	(* PINZA: ASPIRAZIONE/APERTURA CHIUSURA *)
	IF ManCmdJHomeTRIG AND MachinePalletizer_TF.Modules^.AX_J.CmdExe.Code = CmdNOP THEN
		ManCmdJHomeTRIG := FALSE;
	END_IF
	IF MachinePalletizer_TF.ManCmd^.Pinza.ApriPinza THEN
		TFParametersArrayClear(ADR(ParametersArray));
		ParametersArray.Parameters[0] := '1';
		ParametersArray.Parameters[1] := '10';
		TFCommandSend(CmdMAN,ParametersArray,MachinePalletizer_TF.Modules^.Pinza.Cmd);
		MachinePalletizer_TF.ManCmd^.Pinza.ApriPinza := FALSE;
	END_IF
	IF MachinePalletizer_TF.ManCmd^.Pinza.ChiudiPinza THEN
		TFParametersArrayClear(ADR(ParametersArray));
		ParametersArray.Parameters[0] := '1';
		ParametersArray.Parameters[1] := '11';
		MachinePalletizer_TF.ManCmd^.Pinza.ChiudiPinza := FALSE;
		TFCommandSend(CmdMAN,ParametersArray,MachinePalletizer_TF.Modules^.Pinza.Cmd);
	END_IF
	IF MachinePalletizer_TF.ManCmd^.Pinza.SbloccoPinza THEN
		TFParametersArrayClear(ADR(ParametersArray));
		ParametersArray.Parameters[0] := '1';
		ParametersArray.Parameters[1] := '20';
		MachinePalletizer_TF.ManCmd^.Pinza.SbloccoPinza:= FALSE;
		TFCommandSend(CmdMAN,ParametersArray,MachinePalletizer_TF.Modules^.Pinza.Cmd);
	END_IF
	IF MachinePalletizer_TF.ManCmd^.Pinza.BloccoPinza THEN
		TFParametersArrayClear(ADR(ParametersArray));
		ParametersArray.Parameters[0] := '1';
		ParametersArray.Parameters[1] := '21';
		MachinePalletizer_TF.ManCmd^.Pinza.BloccoPinza:= FALSE;
		TFCommandSend(CmdMAN,ParametersArray,MachinePalletizer_TF.Modules^.Pinza.Cmd);
	END_IF
	IF MachinePalletizer_TF.ManCmd^.Pinza.AttivazioneVuotoFaldeDX THEN
		TFParametersArrayClear(ADR(ParametersArray));
		ParametersArray.Parameters[0] := '1';
		ParametersArray.Parameters[1] := '30';
		MachinePalletizer_TF.ManCmd^.Pinza.AttivazioneVuotoFaldeDX := FALSE;
		TFCommandSend(CmdMAN,ParametersArray,MachinePalletizer_TF.Modules^.Pinza.Cmd);
	END_IF
	IF MachinePalletizer_TF.ManCmd^.Pinza.DisattivazioneVuotoFaldeDX THEN
		TFParametersArrayClear(ADR(ParametersArray));
		ParametersArray.Parameters[0] := '1';
		ParametersArray.Parameters[1] := '31';
		MachinePalletizer_TF.ManCmd^.Pinza.DisattivazioneVuotoFaldeDX := FALSE;
		TFCommandSend(CmdMAN,ParametersArray,MachinePalletizer_TF.Modules^.Pinza.Cmd);
	END_IF
	IF MachinePalletizer_TF.ManCmd^.Pinza.AttivazioneVuotoFaldeSX THEN
		TFParametersArrayClear(ADR(ParametersArray));
		ParametersArray.Parameters[0] := '1';
		ParametersArray.Parameters[1] := '40';
		MachinePalletizer_TF.ManCmd^.Pinza.AttivazioneVuotoFaldeSX := FALSE;
		TFCommandSend(CmdMAN,ParametersArray,MachinePalletizer_TF.Modules^.Pinza.Cmd);
	END_IF
	IF MachinePalletizer_TF.ManCmd^.Pinza.DisattivazioneVuotoFaldeSX THEN
		TFParametersArrayClear(ADR(ParametersArray));
		ParametersArray.Parameters[0] := '1';
		ParametersArray.Parameters[1] := '41';
		MachinePalletizer_TF.ManCmd^.Pinza.DisattivazioneVuotoFaldeSX := FALSE;
		TFCommandSend(CmdMAN,ParametersArray,MachinePalletizer_TF.Modules^.Pinza.Cmd);
	END_IF
	IF MachinePalletizer_TF.ManCmd^.Pinza.AttivazioneVuotoDX THEN
		TFParametersArrayClear(ADR(ParametersArray));
		ParametersArray.Parameters[0] := '1';
		ParametersArray.Parameters[1] := '50';
		MachinePalletizer_TF.ManCmd^.Pinza.AttivazioneVuotoDX := FALSE;
		TFCommandSend(CmdMAN,ParametersArray,MachinePalletizer_TF.Modules^.Pinza.Cmd);
	END_IF
//	IF MachinePalletizer_TF.ManCmd^.Pinza.DisattivazioneVuotoDX THEN
//		TFParametersArrayClear(ADR(ParametersArray));
//		ParametersArray.Parameters[0] := '1';
//		ParametersArray.Parameters[1] := '51';
//		MachinePalletizer_TF.ManCmd^.Pinza.DisattivazioneVuotoDX := FALSE;
//		TFCommandSend(CmdMAN,ParametersArray,MachinePalletizer_TF.Modules^.Pinza.Cmd);
//	END_IF
	IF MachinePalletizer_TF.ManCmd^.Pinza.AttivazioneVuotoSX THEN
		TFParametersArrayClear(ADR(ParametersArray));
		ParametersArray.Parameters[0] := '1';
		ParametersArray.Parameters[1] := '60';
		MachinePalletizer_TF.ManCmd^.Pinza.AttivazioneVuotoSX := FALSE;
		TFCommandSend(CmdMAN,ParametersArray,MachinePalletizer_TF.Modules^.Pinza.Cmd);
	END_IF
	IF MachinePalletizer_TF.ManCmd^.Pinza.DisattivazioneVuotoSX THEN
		
		IF Ciclo_Deposito_Lastra.Stato <> ANNULLATO AND NOT EseguitoAllinementoPezziDeposito(*AND MachinePalletizer_TF.Modules^.Pinza.AspirazioneSX^.Out.Attiva_Vuoto AND MachinePalletizer_TF.Modules^.Pinza.StatoPinza.LatoSxPiastrellaInPresa*) THEN
			IF Mission.PPlace > 0 THEN
				//Aggiungo la lastra in deposito e aggiorno lo stato della lastra della lista in modo da contrasegnarla elaborata 
				IF (MachinePalletizerModules.AX_X.Ax^.AxRef^.NcToPlc.ActPos >= WorkArea[Mission.PPlace].X - 300) AND 
					(MachinePalletizerModules.AX_X.Ax^.AxRef^.NcToPlc.ActPos <= WorkArea[Mission.PPlace].X + 300) THEN
					//WorkAreaState[Mission.PPlace].Slab[WorkAreaState[Mission.PPlace].P] 	:= MachinePalletizerModules.Pinza.ElementoInPrelievo^;
					//WorkAreaState[Mission.PPlace].SlabData[WorkAreaState[Mission.PPlace].P] := MachinePalletizerModules.Pinza.DataElement^;
					WorkAreaState[Mission.PPlace].P := WorkAreaState[Mission.PPlace].P +1;
					HMI_NumeroPezziPresentiPostazione[Mission.PPlace] := HMI_NumeroPezziPresentiPostazione[Mission.PPlace] + 1;
					FOR i := 1 TO MAXELEMENTLIST DO
						IF WorkAreaProductionList[Mission.PPlace].PElementList[i].Stato = ELEMENTO_DA_ELABORARE THEN
							WorkAreaProductionList[Mission.PPlace].PElementList[i].Stato := ELEMENTO_ELABORATO; //Dichiaro che l'elemento della lista è stato elaborato
							EXIT;
						END_IF
					END_FOR	
					EseguitoAllinementoPezziDeposito := TRUE;				
				ELSE
					;
				END_IF
				//aggiungo nel prelievo la lastra se è stata rimessa al suo posto
				IF (MachinePalletizerModules.AX_X.Ax^.AxRef^.NcToPlc.ActPos >= WorkArea[Mission.PPick].X - 300) AND 
					(MachinePalletizerModules.AX_X.Ax^.AxRef^.NcToPlc.ActPos <= WorkArea[Mission.PPick].X + 300) THEN
					//WorkAreaState[Mission.PPlace].Slab[WorkAreaState[Mission.PPlace].P] 	:= MachinePalletizerModules.Pinza.ElementoInPrelievo^;
					//WorkAreaState[Mission.PPlace].SlabData[WorkAreaState[Mission.PPlace].P] := MachinePalletizerModules.Pinza.DataElement^;
					WorkAreaState[Mission.PPick].P := WorkAreaState[Mission.PPick].P +1;
					HMI_NumeroPezziPresentiPostazione[Mission.PPick] := HMI_NumeroPezziPresentiPostazione[Mission.PPick] + 1;
					EseguitoAllinementoPezziDeposito := TRUE;	
				ELSE
					;
				END_IF
			END_IF
			
		END_IF
	
		TFParametersArrayClear(ADR(ParametersArray));
		ParametersArray.Parameters[0] := '1';
		ParametersArray.Parameters[1] := '61';
		MachinePalletizer_TF.ManCmd^.Pinza.DisattivazioneVuotoSX := FALSE;
		TFCommandSend(CmdMAN,ParametersArray,MachinePalletizer_TF.Modules^.Pinza.Cmd);
		Ciclo_Prelievo_Lastra.Stato 		:= ANNULLATO;
		Ciclo_Pelievo_Falda.Stato 			:= ANNULLATO;
		Ciclo_Deposito_Lastra.Stato			:= ANNULLATO;
		Ciclo_Deposito_Falda.Stato			:= ANNULLATO;
		Ciclo_Di_Riposo.Stato				:= ANNULLATO;
		Ciclo_Prelievo_Lastra_Depal.Stato 	:= ANNULLATO;
		Ciclo_Deposito_Lastra_Depal.Stato 	:= ANNULLATO;
		Ciclo_Deposito_Falda_Depal.Stato 	:= ANNULLATO;
		ProductOnGripper 					:= KNOPRODUCT;
		Ciclo_Deposito_Falda_Depal.Stato 	:= ANNULLATO;
		
		//Azzero hli apprendimenti e riporto le quote allo stato iniziale
		FOR i:=1 TO MAXAREAPRESENT DO
			WorkAreaState[i].Apprendimento.Z.Lato0.Stato 	:= APPRENDIMENTO_DA_ESEGUIRE;
			WorkAreaState[i].Apprendimento.Z.Lato90.Stato 	:= APPRENDIMENTO_DA_ESEGUIRE;
			WorkAreaState[i].Apprendimento.Z.Lato180.Stato 	:= APPRENDIMENTO_DA_ESEGUIRE;
		END_FOR
		
		StatoMissione 				:= MISSION_STATE_NOP;//Azzero segnalazione a HMI
		WorkAreaManager.State 		:= WAMANAGER_NOP;
		Mission.State 				:= MISSION_STATE_NOP;
		MaterialeDepositatoSuLinea 	:= TRUE;//In questo modo se scarico la mattonella sulla rulliera, lei parte
	END_IF
	IF MachinePalletizer_TF.ManCmd^.Pinza.AttivaTastatori THEN
		TFParametersArrayClear(ADR(ParametersArray));
		ParametersArray.Parameters[0] := '1';
		ParametersArray.Parameters[1] := '70';
		MachinePalletizer_TF.ManCmd^.Pinza.AttivaTastatori := FALSE;
		TFCommandSend(CmdMAN,ParametersArray,MachinePalletizer_TF.Modules^.Pinza.Cmd);
	END_IF
	IF MachinePalletizer_TF.ManCmd^.Pinza.DisattivaTastatori THEN
		TFParametersArrayClear(ADR(ParametersArray));
		ParametersArray.Parameters[0] := '1';
		ParametersArray.Parameters[1] := '71';
		MachinePalletizer_TF.ManCmd^.Pinza.DisattivaTastatori := FALSE;
		TFCommandSend(CmdMAN,ParametersArray,MachinePalletizer_TF.Modules^.Pinza.Cmd);
	END_IF
	IF MachinePalletizer_TF.ManCmd^.Pinza.CalibrazioneOVEM THEN
		TFParametersArrayClear(ADR(ParametersArray));
		MachinePalletizer_TF.ManCmd^.Pinza.CalibrazioneOVEM := FALSE;
		TFCommandSend(CmdHOME,ParametersArray,MachinePalletizer_TF.Modules^.Pinza.Cmd);
	END_IF

	//Posizionamento diretto pinza
	IF MachinePalletizer_TF.ManCmd^.PosizionamentoPinza0 THEN
		TFParametersArrayClear(ADR(ParametersArray));
		ParametersArray.Parameters[0] := '100';
		ParametersArray.Parameters[1] := '13';
		MachinePalletizer_TF.Modules^.AX_J.AxisPar^.Quota_Destinazione := 0;
		TFCommandSend(CmdMAN,ParametersArray,MachinePalletizer_TF.Modules^.AX_J.Cmd);
		MachinePalletizer_TF.ManCmd^.PosizionamentoPinza0 := FALSE;
	END_IF
	IF MachinePalletizer_TF.ManCmd^.PosizionamentoPinza90 THEN
		TFParametersArrayClear(ADR(ParametersArray));
		ParametersArray.Parameters[0] := '100';
		ParametersArray.Parameters[1] := '13';
		MachinePalletizer_TF.Modules^.AX_J.AxisPar^.Quota_Destinazione := 90;
		TFCommandSend(CmdMAN,ParametersArray,MachinePalletizer_TF.Modules^.AX_J.Cmd);
		 MachinePalletizer_TF.ManCmd^.PosizionamentoPinza90 := FALSE;
	END_IF
	IF MachinePalletizer_TF.ManCmd^.PosizionamentoPinza180 THEN
		TFParametersArrayClear(ADR(ParametersArray));
		ParametersArray.Parameters[0] := '100';
		ParametersArray.Parameters[1] := '13';
		MachinePalletizer_TF.Modules^.AX_J.AxisPar^.Quota_Destinazione := 180;
		TFCommandSend(CmdMAN,ParametersArray,MachinePalletizer_TF.Modules^.AX_J.Cmd);
		MachinePalletizer_TF.ManCmd^.PosizionamentoPinza180 := FALSE;
	END_IF
	
	IF ManCmdXHomeTRIG AND 
		MachinePalletizer_TF.Modules^.AX_X.CmdExe.Code = CmdNOP THEN
		ManCmdXHomeTRIG := FALSE;
		MachinePalletizer_TF.ManCmd^.X.Home:= FALSE;
	END_IF
	IF ManCmdYHomeTRIG AND 
		MachinePalletizer_TF.Modules^.AX_Y.CmdExe.Code = CmdNOP THEN
		ManCmdYHomeTRIG := FALSE;
		MachinePalletizer_TF.ManCmd^.Y.Home:= FALSE;
	END_IF
	IF ManCmdZHomeTRIG AND 
		MachinePalletizer_TF.Modules^.AX_Z.CmdExe.Code = CmdNOP THEN
		ManCmdZHomeTRIG := FALSE;
		MachinePalletizer_TF.ManCmd^.Z.Home:= FALSE;
	END_IF
	IF ManCmdJHomeTRIG AND 
		MachinePalletizer_TF.Modules^.AX_J.CmdExe.Code = CmdNOP THEN
		ManCmdJHomeTRIG := FALSE;
		MachinePalletizer_TF.ManCmd^.J.Home:= FALSE;
	END_IF
	
END_IF
END_ACTION

ACTION _06_ScriviOutput:
(* Control Word OVEM *)
O_ControlWordOVEM_1 := MachinePalletizerModules.Pinza.AspirazioneDX1^.Out.ControlWord;
O_ControlWordOVEM_2 := MachinePalletizerModules.Pinza.AspirazioneSX1^.Out.ControlWord;

O_ControlWordOVEM_12 := MachinePalletizerModules.Pinza.AspirazioneDX2^.Out.ControlWord;
O_ControlWordOVEM_22 := MachinePalletizerModules.Pinza.AspirazioneSX2^.Out.ControlWord;

(* Configurazione Porte Ciabatta Pinza *)

{info 'TODO:SISTEMARE IO PINZA'}	

//Q_K517[22] := 1; //Configurazione pin 2 e pin 4 come uscite porta X1.0
//Q_K517[23] := 1; //Configurazione pin 2 e pin 4 come uscite porta X1.1
//Q_K517[24] := 1; //Configurazione pin 2 e pin 4 come uscite porta X1.2
Q_K517[25] := 1; //Configurazione pin 2 e pin 4 come uscite porta X1.3
//Q_K517[26] := 1; //Configurazione pin 2 e pin 4 come uscite porta X1.4
//Q_K517[27] := 1; //Configurazione pin 2 e pin 4 come uscite porta X1.5
Q_K517[28] := 1; //Configurazione pin 2 e pin 4 come uscite porta X1.6
Q_K517[29] := 1; //Configurazione pin 2 e pin 4 come uscite porta X1.7

//Q_K517[2].0 //Comando X1.0 pin 4
//Q_K517[2].1 //Comando X1.1 pin 4
//Q_K517[2].2 //Comando X1.2 pin 4
//Q_K517[2].3 //Comando X1.3 pin 4
//Q_K517[2].4 //Comando X1.4 pin 4
//Q_K517[2].5 //Comando X1.5 pin 4
//Q_K517[2].6 //Comando X1.6 pin 4
//Q_K517[2].7 //Comando X1.7 pin 4
///------------------------------//
//Q_K517[3].0 //Comando X1.0 pin 2
//Q_K517[3].1 //Comando X1.1 pin 2
//Q_K517[3].2 //Comando X1.2 pin 2
//Q_K517[3].3 //Comando X1.3 pin 2
//Q_K517[3].4 //Comando X1.4 pin 2
//Q_K517[3].5 //Comando X1.5 pin 2
//Q_K517[3].6 //Comando X1.6 pin 2
//Q_K517[3].7 //Comando X1.7 pin 2

Q_K517[2].3 := MachinePalletizerModules.Pinza.AspirazioneFaldaDX^.OUT.ActivationOutput;
Q_K517[2].6 := MachinePalletizerModules.Pinza.CilindroSbloccoBascolante^.OUT.ActivationOutput;
Q_K517[2].7 := MachinePalletizerModules.Pinza.CilindroSbloccoRotazione^.OUT.ActivationOutput;

//Q_J17[3].7 := MachinePalletizerModules.Pinza.CilindroTasteggio^.OUT.ActivationOutput;

LetturaFTCPinza0_1 		:= MachinePalletizerModules.Pinza.StatoPinza.LetturaFTC0;
LetturaFTCPinza180_1 	:= MachinePalletizerModules.Pinza.StatoPinza.LetturaFTC180;
LetturaFTCPinza0_2 		:= MachinePalletizerModules.Pinza.StatoPinza.LetturaFTC0_2;
LetturaFTCPinza180_2 	:= MachinePalletizerModules.Pinza.StatoPinza.LetturaFTC180_2;

(* ******************************************************************************************************** *)
(* OUTPUT Transfer *)
(* ******************************************************************************************************** *)

(* Pallet and Layer stacks state *)
PalletStackEmpty 												:= MachinePalletizer_TF.PalletStackEmpty;
LayerStackEmpty 												:= MachinePalletizer_TF.LayerStackEmpty;
AllWABusy 														:= MachinePalletizer_TF.AllWABusy;

(* Machine Palletizer *)
O_ResetACKAzionamenti 	:= I_StartCicloPal OR MachinePalletizerGatesAccess.GateAccessConsolle.ErrAckDriver;// OR MachinePalletizerGatesAccess.GateAccess2.ErrAckDriver;// OR MachinePalletizerLGV.ErrAckDriver;
O_AbilitazioneMarcia	:= MachinePalletizer_TF.OUT.PowerActive;


O_SirenaAllarmiPal		:= MachinePalletizer_TF.OUT.StartHorn OR MachinePalletizer_TF.OUT.Horn OR (MachinePalletizer_TF.OUT.Warning AND MachinePalletizer_TF.OUT.ClockSegnalazioniAlternato AND NOT MachinePalletizer_TF.OUT.ResetSirenaSegnalazioni);// OR (I_Trasporti_GEN_GLOBAL_ALARM_STOP AND MachinePalletizer_TF.OUT.ClockSegnalazioni);

O_LampadaAutomaticoPal	:= MachinePalletizer_TF.OUT.Run;

O_LampadaAllarmiPal		:= (MachinePalletizer_TF.OUT.Error AND MachinePalletizer_TF.OUT.ClockSegnalazioni) OR
							MachinePalletizer_TF.OUT.Error;
							
																	
O_Reset_Plc_Sicurezza := I_StartCicloPal OR 
						MachinePalletizerGatesAccess.GateAccessConsolle.ErrAck OR
						MachinePalletizerGatesAccess.GateAccessPS306.ErrAck OR
						MachinePalletizerGatesAccess.GateAccessPS307.ErrAck OR
						MachinePalletizerGatesAccess.GateAccessPS308.ErrAck OR
						MachinePalletizerGatesAccess.GateAccessPS309.ErrAck;


O_LampadaPulsanteCicloPalConsolle:= MachinePalletizer_TF.OUT.Run OR 
									(ResetNecessarioCentralinaSafety AND MachinePalletizer_TF.OUT.ClockSegnalazioni) ;
O_LampadaPulsanteMarciaPalConsolle := I_MarciaOK AND (MachinePalletizerModules.AX_X.Ax^.Status.PowerActive AND 
													MachinePalletizerModules.AX_Y.Ax^.Status.PowerActive AND 
													MachinePalletizerModules.AX_Z.Ax^.Status.PowerActive AND 
													MachinePalletizerModules.AX_J.Ax^.Status.PowerActive) OR 
										((I_MarciaOK AND NOT(MachinePalletizerModules.AX_X.Ax^.Status.PowerActive AND 
														MachinePalletizerModules.AX_Y.Ax^.Status.PowerActive AND 
														MachinePalletizerModules.AX_Z.Ax^.Status.PowerActive AND 
														MachinePalletizerModules.AX_J.Ax^.Status.PowerActive) OR
										(I_SafetyStateEmergenze_Generali <> 1 OR 
                                          I_SafetyStateEmergenza_PS306_307 <> 1 OR
                                          I_SafetyStateEmergenza_PS308_309 <> 1)) AND MachinePalletizer_TF.OUT.ClockSegnalazioni)AND NOT ResetNecessarioCentralinaSafety;

(* Gates Access *)
O_LampadaRichiestaIngressoPal	:= (MachinePalletizerGatesAccess.GateAccessConsolle.AccessLamp OR 
									MachinePalletizerGatesAccess.GateAccessPS306.AccessLamp OR
									MachinePalletizerGatesAccess.GateAccessPS307.AccessLamp OR 
									MachinePalletizerGatesAccess.GateAccessPS308.AccessLamp OR 
									MachinePalletizerGatesAccess.GateAccessPS309.AccessLamp OR
									(NOT I_BarrierePallettizzatoreOK AND MachinePalletizer_TF.OUT.ClockSegnalazioni))AND NOT ResetNecessarioCentralinaSafety;

O_LampadaPulsanteRichiestaIngressoConsolle := MachinePalletizerGatesAccess.GateAccessConsolle.AccessLamp OR 
											((I_BarrierePallettizzatoreOK <> 1 AND MachinePalletizer_TF.OUT.ClockSegnalazioni) AND NOT ResetNecessarioCentralinaSafety);
									
O_LampadaPulsanteRichiestaIngressoPS306 := MachinePalletizerGatesAccess.GateAccessPS306.AccessLamp OR 
											((NOT I_BarrierePallettizzatoreOK AND MachinePalletizer_TF.OUT.ClockSegnalazioni) AND NOT ResetNecessarioCentralinaSafety);

O_LampadaPulsanteRichiestaIngressoPS307 := MachinePalletizerGatesAccess.GateAccessPS307.AccessLamp OR 
											((NOT I_BarrierePallettizzatoreOK AND MachinePalletizer_TF.OUT.ClockSegnalazioni) AND NOT ResetNecessarioCentralinaSafety);

O_LampadaPulsanteRichiestaIngressoPS308 := MachinePalletizerGatesAccess.GateAccessPS308.AccessLamp OR 
											((NOT I_BarrierePallettizzatoreOK AND MachinePalletizer_TF.OUT.ClockSegnalazioni) AND NOT ResetNecessarioCentralinaSafety);

O_LampadaPulsanteRichiestaIngressoPS309 := MachinePalletizerGatesAccess.GateAccessPS309.AccessLamp OR 
											((NOT I_BarrierePallettizzatoreOK AND MachinePalletizer_TF.OUT.ClockSegnalazioni) AND NOT ResetNecessarioCentralinaSafety);
									
//******************** SCHEDA OUT AP201.4
O_AP201_4[1]	:= O_SirenaAllarmiPal;				
O_AP201_4[2]	:= O_LampadaAutomaticoPal;			
O_AP201_4[3]	:= O_LampadaAllarmiPal;				
O_AP201_4[4]	:= O_LampadaRichiestaIngressoPal;
O_AP201_4[5]	:= O_ConsensoVeicolo[1];						
O_AP201_4[6]	:= O_ConsensoVeicolo[2];						
O_AP201_4[7]	:= O_ConsensoVeicolo[3];						
O_AP201_4[8]	:= O_ConsensoVeicolo[4];						
O_AP201_4[9]	:= O_LampadaPulsanteCicloPalConsolle; 			
O_AP201_4[10]	:= O_LampadaPulsanteRichiestaIngressoConsolle; 	
O_AP201_4[11]	:= O_LampadaPulsanteMarciaPalConsolle;			
O_AP201_4[12]	:= O_LampadaPulsanteRichiestaIngressoPS306; 	
O_AP201_4[13]	:= O_LampadaPulsanteRichiestaIngressoPS307;		
O_AP201_4[14]	:= O_LampadaPulsanteRichiestaIngressoPS308; 	
O_AP201_4[15]	:= O_LampadaPulsanteRichiestaIngressoPS309;		
O_AP201_4[16]	:= FALSE; 										
											
//******************** SCHEDA OUT SAFETY AP201.5											
O_AP201_5;											
//O_MarciaPal	: BOOL; // CH1=											
//FREE			: BOOL; // CH2=												
//FREE			: BOOL; // CH3=												
//FREE			: BOOL; // CH4=			
									
//******************** SCHEDA OUT AP201.6												
O_AP201_6[1]	:= O_LampadaIngressoVietatoPS306; 												
O_AP201_6[2]	:= O_LampadaIngressoVietatoPS307; 												
O_AP201_6[3]	:= O_LampadaIngressoVietatoPS308; 												
O_AP201_6[4]	:= O_LampadaIngressoVietatoPS309; 												
O_AP201_6[5]	:= O_ConsensoVeicolo[5];		  												
O_AP201_6[6]	:= O_ConsensoVeicolo[6];														
O_AP201_6[7]	:= O_ConsensoVeicolo[7];														
O_AP201_6[8]	:= O_ConsensoVeicolo[8];														
O_AP201_6[9]	:= FALSE; 																		
O_AP201_6[10]	:= FALSE; 																		
O_AP201_6[11]	:= FALSE; 																		
O_AP201_6[12]	:= FALSE; 																		
O_AP201_6[13]	:= FALSE; 																		
O_AP201_6[14]	:= FALSE; 							
O_AP201_6[15]	:= FALSE; 							
O_AP201_6[16]	:= FALSE; 							


O_XDriveDigitalOutput.1 := O_SbloccoFermoSicurezza; //Sblocco del paracadute -> ingresso 1 del drive X
END_ACTION

ACTION _07_ScriviStatus:
(*Valorizzazione della struttura Status_TF*)

(*Stato Macchina*)
Status_TF.Macchina.Auto					:= MachinePalletizer_TF.IN.Mode.Auto AND MachinePalletizer_TF.CmdExe.Code = CmdDO;
Status_TF.Macchina.Run					:= MachinePalletizer_TF.OUT.Run;
Status_TF.Macchina.Error				:= MachinePalletizer_TF.Error.Code;
Status_TF.Macchina.ErrorExtra			:= MachinePalletizer_TF.Error.ExtraCode;
Status_TF.Macchina.PowerOK				:= MachinePalletizer_TF.IN.PowerOk;
Status_TF.Macchina.EmergencyOK			:= MachinePalletizer_TF.IN.Mode.EmergencyRequest;

(*Stato assi*)	
Status_TF.X.Position 					:= MachinePalletizerModules.AX_X.Ax^.Status.ActPosition;
Status_TF.X.Velocity 					:= MachinePalletizerModules.AX_X.Ax^.Status.ActVelocity;
Status_TF.X.Torque 						:= MachinePalletizerModules.AX_X.Ax^.Status.ActTorque;
Status_TF.X.Error 						:= MachinePalletizerModules.AX_X.Ax^.Status.ErrorID;
Status_TF.X.PowerActive					:= MachinePalletizerModules.AX_X.Ax^.Status.PowerActive;

Status_TF.Y.Position 					:= MachinePalletizerModules.AX_Y.Ax^.Status.ActPosition;
Status_TF.Y.Velocity 					:= MachinePalletizerModules.AX_Y.Ax^.Status.ActVelocity;
Status_TF.Y.Torque 						:= MachinePalletizerModules.AX_Y.Ax^.Status.ActTorque;
Status_TF.Y.Error 						:= MachinePalletizerModules.AX_Y.Ax^.Status.ErrorID;
Status_TF.Y.PowerActive					:= MachinePalletizerModules.AX_Y.Ax^.Status.PowerActive;

Status_TF.Z.Position 					:= MachinePalletizerModules.AX_Z.Ax^.Status.ActPosition;
Status_TF.Z.Velocity 					:= MachinePalletizerModules.AX_Z.Ax^.Status.ActVelocity;
Status_TF.Z.Torque 						:= MachinePalletizerModules.AX_Z.Ax^.Status.ActTorque;
Status_TF.Z.Error 						:= MachinePalletizerModules.AX_Z.Ax^.Status.ErrorID;
Status_TF.Z.PowerActive					:= MachinePalletizerModules.AX_Z.Ax^.Status.PowerActive;

Status_TF.J.Position 					:= MachinePalletizerModules.AX_J.Ax^.Status.ActPosition;
Status_TF.J.Velocity 					:= MachinePalletizerModules.AX_J.Ax^.Status.ActVelocity;
Status_TF.J.Torque 						:= MachinePalletizerModules.AX_J.Ax^.Status.ActTorque;
Status_TF.J.Error 						:= MachinePalletizerModules.AX_J.Ax^.Status.ErrorID;
Status_TF.J.PowerActive					:= MachinePalletizerModules.AX_J.Ax^.Status.PowerActive;

Status_TF.K.Position 					:= 0;//ModuloAsse_K.Ax^.Status.ActPosition;
Status_TF.K.Velocity 					:= 0;//ModuloAsse_K.Ax^.Status.ActVelocity;
Status_TF.K.Torque 						:= 0;//ModuloAsse_K.Ax^.Status.ActTorque;
Status_TF.K.Error 						:= 0;//ModuloAsse_K.Ax^.Status.ErrorID;
Status_TF.K.PowerActive					:= 0;//ModuloAsse_K.Ax^.Status.PowerActive;

(*Stato Moduli*)
//Status_TF.ModAsse_X.Cmd					:= ModuloAsse_X.CmdExe.Code;
//Status_TF.ModAsse_X.CmdCase				:= ModuloAsse_X.CmdExe.CmdCase;
Status_TF.ModAsse_X.Error       		:= MachinePalletizerModules.AX_X.Error.Code;
Status_TF.ModAsse_X.ErrorExtra      	:= MachinePalletizerModules.AX_X.Error.ExtraCode;

//Status_TF.ModAsse_Y.Cmd					:= ModuloAsse_Y.CmdExe.Code;
//Status_TF.ModAsse_Y.CmdCase				:= ModuloAsse_Y.CmdExe.CmdCase;
Status_TF.ModAsse_Y.Error       		:= MachinePalletizerModules.AX_Y.Error.Code;
Status_TF.ModAsse_Y.ErrorExtra      	:= MachinePalletizerModules.AX_Y.Error.ExtraCode;

//Status_TF.ModAsse_Z.Cmd					:= ModuloAsse_Z.CmdExe.Code;
//Status_TF.ModAsse_Z.CmdCase				:= ModuloAsse_Z.CmdExe.CmdCase;
Status_TF.ModAsse_Z.Error       		:= MachinePalletizerModules.AX_Z.Error.Code;
Status_TF.ModAsse_Z.ErrorExtra      	:= MachinePalletizerModules.AX_Z.Error.ExtraCode;

//Status_TF.ModAsse_J.Cmd					:= ModuloAsse_J.CmdExe.Code;
//Status_TF.ModAsse_J.CmdCase				:= ModuloAsse_J.CmdExe.CmdCase;
Status_TF.ModAsse_J.Error       		:= MachinePalletizerModules.AX_J.Error.Code;
Status_TF.ModAsse_J.ErrorExtra      	:= MachinePalletizerModules.AX_J.Error.ExtraCode;

//Status_TF.ModAsse_K.Cmd					:= ModuloAsse_K.CmdExe.Code;
//Status_TF.ModAsse_K.CmdCase				:= ModuloAsse_K.CmdExe.CmdCase;
Status_TF.ModAsse_K.Error       		:= 0;//ModuloAsse_K.Error.Code;
Status_TF.ModAsse_K.ErrorExtra      	:= 0;//ModuloAsse_K.Error.ExtraCode;

//Status_TF.ModAspirazione.Cmd			:= ModuloAspirazione.CmdExe.Code;
//Status_TF.ModAspirazione.CmdCase		:= ModuloAspirazione.CmdExe.CmdCase;
Status_TF.ModAspirazione.Error       	:= MachinePalletizerModules.Pinza.Error.Code;
Status_TF.ModAspirazione.ErrorExtra     := MachinePalletizerModules.Pinza.Error.ExtraCode;

Status_TF.Pinza.Module.Error       	:= MachinePalletizerModules.Pinza.Error.Code;
Status_TF.Pinza.Module.ErrorExtra     := MachinePalletizerModules.Pinza.Error.ExtraCode;


(* Trsferimento a Struttura dati Creo *)
Status.MachineAuto := Status_TF.Macchina.Auto;
Status.MachineError := Status_TF.Macchina.Error;
Status.MachineErrorExtra := Status_TF.Macchina.ErrorExtra;

//Pinza Cilindro Cilindro Aspirazione DX
Status_TF.Pinza.AspirazioneDX.Active 			:= MachinePalletizerModules.Pinza.AspirazioneDX1^.Status.Aspirazione_ON; 
Status_TF.Pinza.AspirazioneDX.Inactive 		:= MachinePalletizerModules.Pinza.AspirazioneDX1^.Status.Aspirazione_OFF; 
Status_TF.Pinza.AspirazioneDX.SensorActive 	:= MachinePalletizerModules.Pinza.AspirazioneDX1^.Status.DepressioneSoglia1_OK; 
Status_TF.Pinza.AspirazioneDX.SensorInactive 	:= NOT MachinePalletizerModules.Pinza.AspirazioneDX1^.Status.DepressioneSoglia1_OK; 

Status_TF.Pinza.AspirazioneDX.Error := ErrBASEOVEM+MachinePalletizerModules.Pinza.AspirazioneDX1^.Status.ErrorID;
IF Status_TF.Pinza.AspirazioneDX.Error <> ErrBASEOVEM THEN 
	Status_TF.Pinza.AspirazioneDX.StatusToHMI := 9;
ELSIF MachinePalletizerModules.Pinza.AspirazioneDX1^.Status.Aspirazione_ON THEN
	Status_TF.Pinza.AspirazioneDX.StatusToHMI := 1;
ELSIF MachinePalletizerModules.Pinza.AspirazioneDX1^.Status.Aspirazione_OFF THEN
	Status_TF.Pinza.AspirazioneDX.StatusToHMI := 2;
END_IF
IF Status_TF.Pinza.AspirazioneDX.Error = ErrBASEOVEM THEN
	Status_TF.Pinza.AspirazioneDX.Error := 0;
END_IF


//Pinza Cilindro Cilindro AspirazioneFalda SX
Status_TF.Pinza.AspirazioneSX.Active 			:= MachinePalletizerModules.Pinza.AspirazioneSX1^.Status.Aspirazione_ON; 
Status_TF.Pinza.AspirazioneSX.Inactive 		:= MachinePalletizerModules.Pinza.AspirazioneSX1^.Status.Aspirazione_OFF; 
Status_TF.Pinza.AspirazioneSX.SensorActive 	:= MachinePalletizerModules.Pinza.AspirazioneSX1^.Status.DepressioneSoglia1_OK; 
Status_TF.Pinza.AspirazioneSX.SensorInactive 	:= NOT MachinePalletizerModules.Pinza.AspirazioneSX1^.Status.DepressioneSoglia1_OK; 

Status_TF.Pinza.AspirazioneSX.Error := ErrBASEOVEM+MachinePalletizerModules.Pinza.AspirazioneSX1^.Status.ErrorID ;
IF Status_TF.Pinza.AspirazioneSX.Error  <> ErrBASEOVEM THEN 
	Status_TF.Pinza.AspirazioneSX.StatusToHMI := 9;
ELSIF MachinePalletizerModules.Pinza.AspirazioneSX1^.Status.Aspirazione_ON THEN
	Status_TF.Pinza.AspirazioneSX.StatusToHMI := 1;
ELSIF MachinePalletizerModules.Pinza.AspirazioneSX1^.Status.Aspirazione_OFF THEN
	Status_TF.Pinza.AspirazioneSX.StatusToHMI := 2;
END_IF
IF Status_TF.Pinza.AspirazioneSX.Error = ErrBASEOVEM THEN
	Status_TF.Pinza.AspirazioneSX.Error := 0;
END_IF

//Pinza Cilindro Cilindro Apertura pinza 
Status_TF.Pinza.CilindroApertura.Active 			:= MachinePalletizerModules.Pinza.CilindroApertura^.Status.Active; 
Status_TF.Pinza.CilindroApertura.Inactive 			:= MachinePalletizerModules.Pinza.CilindroApertura^.Status.Inactive; 
Status_TF.Pinza.CilindroApertura.SensorActive 		:= MachinePalletizerModules.Pinza.CilindroApertura^.IN.PX_Active; 
Status_TF.Pinza.CilindroApertura.SensorInactive 	:= NOT MachinePalletizerModules.Pinza.CilindroApertura^.IN.PX_Inactive; 

Status_TF.Pinza.CilindroApertura.Error := MachinePalletizerModules.Pinza.CilindroApertura^.Status.ErrorID ;
IF Status_TF.Pinza.CilindroApertura.Error  <> 0 THEN 
	Status_TF.Pinza.CilindroApertura.StatusToHMI := 9;
ELSIF MachinePalletizerModules.Pinza.CilindroApertura^.Status.Active THEN
	Status_TF.Pinza.CilindroApertura.StatusToHMI := 1;
ELSIF MachinePalletizerModules.Pinza.CilindroApertura^.Status.Inactive THEN
	Status_TF.Pinza.CilindroApertura.StatusToHMI := 2;
END_IF
IF Status_TF.Pinza.CilindroApertura.Error = 0 THEN
	Status_TF.Pinza.CilindroApertura.Error := 0;
END_IF

//Aspirazione SX2 
Status_TF.Pinza.AspirazioneSX2.Active 			:= MachinePalletizerModules.Pinza.AspirazioneSX2^.Status.Aspirazione_ON; 
Status_TF.Pinza.AspirazioneSX2.Inactive 		:= MachinePalletizerModules.Pinza.AspirazioneSX2^.Status.Aspirazione_OFF; 
Status_TF.Pinza.AspirazioneSX2.SensorActive 	:= MachinePalletizerModules.Pinza.AspirazioneSX2^.Status.DepressioneSoglia1_OK; 
Status_TF.Pinza.AspirazioneSX2.SensorInactive 	:= NOT MachinePalletizerModules.Pinza.AspirazioneSX2^.Status.DepressioneSoglia1_OK; 

Status_TF.Pinza.AspirazioneSX2.Error := ErrBASEOVEM+MachinePalletizerModules.Pinza.AspirazioneSX2^.Status.ErrorID ;
IF Status_TF.Pinza.AspirazioneSX2.Error  <> ErrBASEOVEM THEN 
	Status_TF.Pinza.AspirazioneSX2.StatusToHMI := 9;
ELSIF MachinePalletizerModules.Pinza.AspirazioneSX2^.Status.Aspirazione_ON THEN
	Status_TF.Pinza.AspirazioneSX2.StatusToHMI := 1;
ELSIF MachinePalletizerModules.Pinza.AspirazioneSX2^.Status.Aspirazione_OFF THEN
	Status_TF.Pinza.AspirazioneSX2.StatusToHMI := 2;
END_IF
IF Status_TF.Pinza.AspirazioneSX2.Error = ErrBASEOVEM THEN
	Status_TF.Pinza.AspirazioneSX2.Error := 0;
END_IF
//Aspirazione DX 
Status_TF.Pinza.AspirazioneDX2.Active 			:= MachinePalletizerModules.Pinza.AspirazioneDX2^.Status.Aspirazione_ON; 
Status_TF.Pinza.AspirazioneDX2.Inactive 		:= MachinePalletizerModules.Pinza.AspirazioneDX2^.Status.Aspirazione_OFF; 
Status_TF.Pinza.AspirazioneDX2.SensorActive 	:= MachinePalletizerModules.Pinza.AspirazioneDX2^.Status.DepressioneSoglia1_OK; 
Status_TF.Pinza.AspirazioneDX2.SensorInactive 	:= NOT MachinePalletizerModules.Pinza.AspirazioneDX2^.Status.DepressioneSoglia1_OK; 

Status_TF.Pinza.AspirazioneDX2.Error := ErrBASEOVEM+MachinePalletizerModules.Pinza.AspirazioneDX2^.Status.ErrorID;
IF Status_TF.Pinza.AspirazioneDX2.Error <> ErrBASEOVEM THEN 
	Status_TF.Pinza.AspirazioneDX2.StatusToHMI := 9;
ELSIF MachinePalletizerModules.Pinza.AspirazioneDX2^.Status.Aspirazione_ON THEN
	Status_TF.Pinza.AspirazioneDX2.StatusToHMI := 1;
ELSIF MachinePalletizerModules.Pinza.AspirazioneDX2^.Status.Aspirazione_OFF THEN
	Status_TF.Pinza.AspirazioneDX2.StatusToHMI := 2;
END_IF
IF Status_TF.Pinza.AspirazioneDX.Error = ErrBASEOVEM THEN
	Status_TF.Pinza.AspirazioneDX.Error := 0;
END_IF

//Pinza Cilindro Cilindro Sblocco Rotazione
Status_TF.Pinza.CilindroSbloccoRotazione.Active 			:= MachinePalletizerModules.Pinza.CilindroSbloccoRotazione^.Status.Active; 
Status_TF.Pinza.CilindroSbloccoRotazione.Inactive 			:= MachinePalletizerModules.Pinza.CilindroSbloccoRotazione^.Status.Inactive; 
Status_TF.Pinza.CilindroSbloccoRotazione.SensorActive 		:= MachinePalletizerModules.Pinza.CilindroSbloccoRotazione^.IN.PX_Active; 
Status_TF.Pinza.CilindroSbloccoRotazione.SensorInactive 	:= NOT MachinePalletizerModules.Pinza.CilindroSbloccoRotazione^.IN.PX_Inactive; 

Status_TF.Pinza.CilindroSbloccoRotazione.Error := MachinePalletizerModules.Pinza.CilindroSbloccoRotazione^.Status.ErrorID ;
IF Status_TF.Pinza.CilindroSbloccoRotazione.Error  <> 0 THEN 
	Status_TF.Pinza.CilindroSbloccoRotazione.StatusToHMI := 9;
ELSIF MachinePalletizerModules.Pinza.CilindroSbloccoRotazione^.Status.Active THEN
	Status_TF.Pinza.CilindroSbloccoRotazione.StatusToHMI := 1;
ELSIF MachinePalletizerModules.Pinza.CilindroSbloccoRotazione^.Status.Inactive THEN
	Status_TF.Pinza.CilindroSbloccoRotazione.StatusToHMI := 2;
END_IF
IF Status_TF.Pinza.CilindroSbloccoRotazione.Error = 0 THEN
	Status_TF.Pinza.CilindroSbloccoRotazione.Error := 0;
END_IF

//Pinza Cilindro Cilindro Sblocco Bascolante
Status_TF.Pinza.CilindroSbloccoBascolante.Active 			:= MachinePalletizerModules.Pinza.CilindroSbloccoBascolante^.Status.Active; 
Status_TF.Pinza.CilindroSbloccoBascolante.Inactive 			:= MachinePalletizerModules.Pinza.CilindroSbloccoBascolante^.Status.Inactive; 
Status_TF.Pinza.CilindroSbloccoBascolante.SensorActive 		:= MachinePalletizerModules.Pinza.CilindroSbloccoBascolante^.IN.PX_Active; 
Status_TF.Pinza.CilindroSbloccoBascolante.SensorInactive 	:= NOT MachinePalletizerModules.Pinza.CilindroSbloccoBascolante^.IN.PX_Inactive; 

Status_TF.Pinza.CilindroSbloccoBascolante.Error := MachinePalletizerModules.Pinza.CilindroSbloccoBascolante^.Status.ErrorID ;
IF Status_TF.Pinza.CilindroSbloccoBascolante.Error  <> 0 THEN 
	Status_TF.Pinza.CilindroSbloccoBascolante.StatusToHMI := 9;
ELSIF MachinePalletizerModules.Pinza.CilindroSbloccoBascolante^.Status.Active THEN
	Status_TF.Pinza.CilindroSbloccoBascolante.StatusToHMI := 1;
ELSIF MachinePalletizerModules.Pinza.CilindroSbloccoBascolante^.Status.Inactive THEN
	Status_TF.Pinza.CilindroSbloccoBascolante.StatusToHMI := 2;
END_IF
IF Status_TF.Pinza.CilindroSbloccoBascolante.Error = 0 THEN
	Status_TF.Pinza.CilindroSbloccoBascolante.Error := 0;
END_IF


//Trasferisco segnalazione stato a HMI
IF Mission.State > 0 THEN
	StatoMissione := Mission.State;
ELSE
	StatoMissione := MISSION_STATE_NOP;
END_IF
//Aggiorno valori stato postazione
FOR i:=1 TO MAXAREAPRESENT DO
	HMI_Stato_Postazione[i].Abilitata 			:= WorkArea[i].Enable; 
	HMI_Stato_Postazione[i].CodiceFormatura		:= WorkAreaState[i].F;
	HMI_Stato_Postazione[i].CodiceLavorazione	:= WorkAreaState[i].Code;
	HMI_Stato_Postazione[i].LGV_Req				:= WorkAreaState[i].LGV_Req;
	HMI_Stato_Postazione[i].NPezzi				:= WorkAreaState[i].P -1;
	HMI_Stato_Postazione[i].ProgressiveNr		:= TO_UDINT(WorkAreaState[i].ID);	
	HMI_Stato_Postazione[i].Stato 				:= WorkAreaState[i].State;
	HMI_Stato_Postazione[i].TipologiaPostazione := WorkArea[i].Typology;
	HMI_Stato_Postazione[i].TipologiaSupporto 	:= WorkAreaState[i].Supporto.Tipologia;
	IF Status_TF.Macchina.Auto THEN
		HMI_NumeroPezziPresentiPostazione[i] := MAX(0,WorkAreaState[i].P-1);
	END_IF
END_FOR

//STATO SICUREZZE
HMI_Status_FungiPal_OK 			:= I_SafetyStateEmergenza_PS306_307 = 1 AND I_SafetyStateEmergenza_PS308_309 = 1;
HMI_Status_FungoGenerale_OK 	:= I_SafetyStateEmergenze_Generali = 1;
HMI_Status_Funghi_OK 			:= HMI_Status_FungiPal_OK AND
                                   HMI_Status_FungoGenerale_OK;
 	    
HMI_Status_BarrierDXPal_OK 			:= I_SafetyStateBarrierDXPal  = 1;	
HMI_Status_BarrierSXPal_OK 			:= I_SafetyStateBarrierSXPal  = 1;				
HMI_Status_BarrierCentroDXPal_OK	:= I_SafetyStateBarrierCentroDXPal  = 1;		
HMI_Status_BarrierCentroSXPal_OK	:= I_SafetyStateBarrierCentroSXPal  = 1;		
HMI_Status_StateBarrierKarv_OK    	:= I_SafetyStateBarrierKarv  = 1;				

HMI_Status_BarrieraPall_OK			:= HMI_Status_BarrierDXPal_OK AND 		   
                                       HMI_Status_BarrierSXPal_OK AND 		   
                                       HMI_Status_BarrierCentroDXPal_OK AND
                                       HMI_Status_BarrierCentroSXPal_OK AND
									   HMI_Status_StateBarrierKarv_OK;
(*VISUALIZZAZIONE I/O SU PREMIUM HMI*)
HMI_AP200_2 := I_AP200_2;  	
HMI_AP200_3 := I_AP200_3;  
HMI_AP200_4 := I_AP200_4;  
HMI_AP200_5 := I_AP200_5;  
HMI_AP200_6	:= I_AP200_6;	 
HMI_AP200_7	:= I_AP200_7;	 
HMI_AP200_8 := I_AP200_8;  
HMI_AP200_9	:= I_AP200_9;	 
HMI_AP200_10:= I_AP200_10; 
HMI_AP201_2	:= I_AP201_2;	 
HMI_AP201_4 := O_AP201_4;  
HMI_AP201_5	:= I_AP201_5;	 
HMI_AP201_6 := O_AP201_6;  
HMI_AP201_3 := I_AP201_3;  
HMI_AP202_2	:= I_AP202_2;	 
HMI_AP202_3	:= I_AP202_3;	 
HMI_AP202_5	:= I_AP202_5;	 
HMI_AP202_6	:= I_AP202_6;	 

HMI_DepressioneOVEM_DX1 := Pinza.Ovem1.Status.ValoreDepressioneIstantanea;
HMI_DepressioneOVEM_DX2 := Pinza.Ovem12.Status.ValoreDepressioneIstantanea;

HMI_DepressioneOVEM_SX1 := Pinza.Ovem2.Status.ValoreDepressioneIstantanea;
HMI_DepressioneOVEM_SX2 := Pinza.Ovem22.Status.ValoreDepressioneIstantanea;

{info 'TODO:SISTEMARE IO PINZA X HMI'}	
//HMI_DepressioneOVEM_SX1 
////
//HMI_LetturaFTCPinza0_1 	
//HMI_LetturaFTCPinza180_1
//HMI_DepressioneOVEM_SX2 
////CIABATTA 516	
//HMI_DepressioneOVEM_DX1 
//HMI_DepressioneOVEM_DX2 
//HMI_LetturaFTCPinza0_2	
//HMI_LetturaFTCPinza180_2
//HMI_K516_51 			
//HMI_K516_52 			
//HMI_K516_61 			
//HMI_K516_62 			
//HMI_K516_71 			
//HMI_K516_72 			
//HMI_K516_81 			
//HMI_K516_82 			
////CIABATTA 517	
//HMI_K517_11  			
//HMI_K517_12  			
//HMI_K517_21  			
//HMI_K517_22  			
//HMI_K517_31  			
//HMI_K517_32  			
//HMI_K517_41  			
//HMI_K517_42  			
//HMI_K517_51 			
//HMI_K517_52 			
//HMI_K517_61 			
//HMI_K517_62 			
//HMI_K517_71 			
//HMI_K517_72 			
//HMI_K517_81 			
//HMI_K517_82
END_ACTION

ACTION _08_DataLogger_ACT:
// INIT - Assegnazione codici in verifica da formature - Verifico su quale fomatura è associato l codice i-esimo e scrivo la formatura associata nell'array di riferimento.
// Non posso avere duplicazioni in quanto è il supervisore a verificare che tutto sia concorde
// L'Array ottenuto, rappresenta la sequenza delle formature in cui ho un codice i-esimo
// es: formatura 1 con codici assegnati 7 e 10, formatura 3 con codicie da 1 a 4 pieni e formatura 4 con codice 15 -> 3,3,3,3,0,0,1,0,0,1,0,0,0,0,4.....
// Step 1 - cancello struttura
FOR k := 1 TO MAXFORMINGCODE DO
	DATA_LOGGER.Formign_ID_Active_Code[k] := 0;
END_FOR
// Step 2 - assegno valori attuali
FOR i := 1 TO MAXFORMING DO
	FOR k := 1 TO MAXFORMINGCODE DO 
		IF Forming[i].Code[k] <> 0 and Forming[i].Code[k] <> -1 THEN
			DATA_LOGGER.Formign_ID_Active_Code[k] := UINT_TO_INT(i);
		END_IF
	END_FOR
END_FOR

DLogger(Auto_GENERAL :=  MachinePalletizer_TF.CmdExe.Code = CmdDO, 
		Alarm_GENERAL := MachinePalletizer_TF.OUT.Error AND MachinePalletizer_TF.CmdExe.Code <> CmdDO,Man_GENERAL := MachinePalletizer_TF.IN.Mode.Man AND Status.MachineError = 0, 
		RI_GENERAL := MachinePalletizerGatesAccess.GateAccessConsolle.AccesActive (*OR MachinePalletizerGatesAccess.GateAccess2.AccesActive*),// OR MachinePalletizerLGV.LGVAccesActive, 
		Global_Reset := DLOG_Cmd_ResetCounter, 
		Daily_Reset := INT_TO_WORD(DLOG_Day_Reset), Weekly_Reset := INT_TO_WORD(DLOG_Week_Reset),
		Alarm_Reset := DLOG_Cmd_Alarm_reset,
		StoricoFile := DLOG_SaveDataOnReset,
		FilePath := 'C:\Logger\LogFile.txt',
		Channel := Channels);
		
Clogger(Global_Reset := CLOG_Global_reset,
		Daily_Reset := INT_TO_WORD(DLOG_Day_Reset), Weekly_Reset := INT_TO_WORD(DLOG_Week_Reset),
		Alarm_Reset := DLOG_Cmd_Alarm_reset,
		StoricoFile := DLOG_SaveDataOnReset,
		FilePath := 'C:\Logger\LogCounter.txt',
		Enable_Log_HMI := dlogger.Enable_Log_HMI,
		NumeroCanaliDatiProd := 16,
		Channel := Counters);
		
// Impostazione canali DataLogger
// Canale 1 - Mancanza pallet vuoti in ciclo automatico
Channels[0].Enable := TRUE;
Channels[0].Nome := 'Mancanza pallet vuoti in ciclo automatico';
Channels[0].Signal := PalletStackEmpty = 1 AND MachinePalletizer_TF.WorkAreaManager^.State = WAMANAGER_NOP AND MachinePalletizer_TF.CmdExe.Code = CmdDO;
Channels[0].Daily_Reference_Total := DLogger.Stat_Auto.Daily_Counter_State;
Channels[0].Weekly_Reference_Total := DLogger.Stat_Auto.Weekly_Counter_State;

// Canale 2 - Nessuna missione attiva su pallettizzatore in ciclo automatico
Channels[1].Enable := TRUE;
Channels[1].Nome := 'Nessuna missione attiva su pallettizzatore in ciclo automatico';
Channels[1].Signal := MachinePalletizer_TF.WorkAreaManager^.State = WAMANAGER_NOP AND MachinePalletizer_TF.CmdExe.Code = CmdDO;
Channels[1].Daily_Reference_Total := DLogger.Stat_Auto.Daily_Counter_State;
Channels[1].Weekly_Reference_Total := DLogger.Stat_Auto.Weekly_Counter_State;

// Canale 3 - Richiesta ingresso navetta su richiesta ingresso generale
(*Channels[2].Enable := TRUE;
Channels[2].Nome := 'Richiesta ingresso navetta su richiesta ingresso generale';
Channels[2].Signal := MachinePalletizerLGV.LGVAccesActive;
Channels[2].Daily_Reference_Total := DLogger.Stat_RI.Daily_Counter_State;
Channels[2].Weekly_Reference_Total := DLogger.Stat_RI.Weekly_Counter_State;
*)
// Canale 4 - Tutte le WA impegnate sul totale di automatico
Channels[3].Enable := TRUE;
Channels[3].Nome := 'Tutte le WA impegnate sul totale di automatico';
Channels[3].Signal := MachinePalletizer_TF.AllWABusy = 1 AND MachinePalletizer_TF.CmdExe.Code = CmdDO;
Channels[3].Daily_Reference_Total := DLogger.Stat_Auto.Daily_Counter_State;
Channels[3].Weekly_Reference_Total := DLogger.Stat_Auto.Weekly_Counter_State;

// Canale 5 - Tutte le WA impegnate sul totale di missione nulla
Channels[4].Enable := TRUE;
Channels[4].Nome := 'Tutte le WA impegnate sul totale di missione nulla';
Channels[4].Signal := MachinePalletizer_TF.AllWABusy = 1 AND MachinePalletizer_TF.CmdExe.Code = CmdDO;
Channels[4].Daily_Reference_Total := Channels[1].Daily_Counter_State;
Channels[4].Weekly_Reference_Total := Channels[1].Weekly_Counter_State;


////////////////////////////////////////////////////////////////////////////////////////////////////////
////////////////////////////////////////////////////////////////////////////////////////////////////////
// Impostazione canali CounterLogger
// Canale 1 - Totale pacchi prelevati - riservato non resettabile da operatore
Counters[0].Enable := TRUE;
Counters[0].Nome := 'Totale pacchi prelevati da ribaltino';
Counters[0].Signal := MachinePalletizer_TF.CmdExe.Code = CmdDO AND PaccoPresoXDataLogger;
Counters[0].Enable_Reset_Storico := FALSE;
Counters[0].ResetCounter := FALSE;
Counters[0].Daily_Reference_Total := 100;
Counters[0].Weekly_Reference_Total := 100;


// Canale 2 - Totale Pacchi parziali
Counters[1].Enable := TRUE;
Counters[1].Nome := 'Totale pacchi prelevati da ribaltino - parziale';
Counters[1].Signal := MachinePalletizer_TF.CmdExe.Code = CmdDO AND PaccoPresoXDataLogger;
Counters[1].Enable_Reset_Storico := FALSE;
Counters[1].ResetCounter := DATA_LOGGER.Reset_Operatore;
Counters[1].Daily_Reference_Total := 100;
Counters[1].Weekly_Reference_Total := 100;
Counters[1].Enable_Reset_Dopo_Salvataggio := TRUE;

(*
// Verifica segnale codice assegnato
FOR i := 1 TO 15 DO
	Counters[i + 1].Signal := MachinePalletizer_TF.CmdExe.Code = CmdDO AND PaccoPresoXDataLogger 
				AND WorkPickPointState[Mission.PPick].Code = (*Forming[DATA_LOGGER.Formign_ID_Active_Code[i]].Code[i]*) i AND WorkPickPointState[Mission.PPick].Code <> 0;
END_FOR
*)
// Conteggio riferimento pacchi parziali - somma di tutti i pacchi contati atualmente dopo reset parziale
TotalePacchiParziali := 0;
FOR i := 2 TO 16 DO
	TotalePacchiParziali := TotalePacchiParziali + Counters[I].Daily_Periodic_Counter_State;
END_FOR

// Canale 3 - Totale pacchi primo codice - parziale
Counters[2].Enable := TRUE;
Counters[2].Nome := CONCAT(STR1:= 'Primo codice - parziale, VALORE -> ', STR2 := INT_TO_STRING(1));
Counters[2].Enable_Reset_Storico := FALSE;
Counters[2].ResetCounter := DATA_LOGGER.Reset_Operatore;
Counters[2].Daily_Reference_Total := Counters[1].Daily_Counter_State;
Counters[2].Weekly_Reference_Total := Counters[1].Weekly_Counter_State;
Counters[2].Periodic_Reference_Total := TotalePacchiParziali;
Counters[2].Enable_Reset_Dopo_Salvataggio := TRUE;

// Canale 3 - Totale pacchi secondo codice - parziale
Counters[3].Enable := TRUE;
Counters[3].Nome := CONCAT(STR1:= 'Secondo codice - parziale, VALORE -> ', STR2 := INT_TO_STRING(2));
Counters[3].Enable_Reset_Storico := FALSE;
Counters[3].ResetCounter := DATA_LOGGER.Reset_Operatore;
Counters[3].Daily_Reference_Total := Counters[1].Daily_Counter_State;
Counters[3].Weekly_Reference_Total := Counters[1].Weekly_Counter_State;
Counters[3].Periodic_Reference_Total := TotalePacchiParziali;
Counters[3].Enable_Reset_Dopo_Salvataggio := TRUE;

// Canale 4 - Totale pacchi terzo codice - parziale
Counters[4].Enable := TRUE;
Counters[4].Nome := CONCAT(STR1:= 'Terzo codice - parziale, VALORE -> ', STR2 := INT_TO_STRING(3));
Counters[4].Enable_Reset_Storico := FALSE;
Counters[4].ResetCounter := DATA_LOGGER.Reset_Operatore;
Counters[4].Daily_Reference_Total := Counters[1].Daily_Counter_State;
Counters[4].Weekly_Reference_Total := Counters[1].Weekly_Counter_State;
Counters[4].Periodic_Reference_Total := TotalePacchiParziali;
Counters[4].Enable_Reset_Dopo_Salvataggio := TRUE;

// Canale 5 - Totale pacchi quarto codice - parziale
Counters[5].Enable := TRUE;
Counters[5].Nome := CONCAT(STR1:= 'Quarto codice - parziale, VALORE -> ', STR2 := INT_TO_STRING(4));
Counters[5].Enable_Reset_Storico := FALSE;
Counters[5].ResetCounter := DATA_LOGGER.Reset_Operatore;
Counters[5].Daily_Reference_Total := Counters[1].Daily_Counter_State;
Counters[5].Weekly_Reference_Total := Counters[1].Weekly_Counter_State;
Counters[5].Periodic_Reference_Total := TotalePacchiParziali;
Counters[5].Enable_Reset_Dopo_Salvataggio := TRUE;

// Canale 6 - Totale pacchi quinto codice - parziale
Counters[6].Enable := TRUE;
Counters[6].Nome := CONCAT(STR1:= 'Quinto codice - parziale, VALORE -> ', STR2 := INT_TO_STRING(5));
Counters[6].Enable_Reset_Storico := FALSE;
Counters[6].ResetCounter := DATA_LOGGER.Reset_Operatore;
Counters[6].Daily_Reference_Total := Counters[1].Daily_Counter_State;
Counters[6].Weekly_Reference_Total := Counters[1].Weekly_Counter_State;
Counters[6].Periodic_Reference_Total := TotalePacchiParziali;
Counters[6].Enable_Reset_Dopo_Salvataggio := TRUE;

// Canale 7 - Totale pacchi sesto codice - parziale
Counters[7].Enable := TRUE;
Counters[7].Nome := CONCAT(STR1:= 'Sesto codice - parziale, VALORE -> ', STR2 := INT_TO_STRING(6));
Counters[7].Enable_Reset_Storico := FALSE;
Counters[7].ResetCounter := DATA_LOGGER.Reset_Operatore;
Counters[7].Daily_Reference_Total := Counters[1].Daily_Counter_State;
Counters[7].Weekly_Reference_Total := Counters[1].Weekly_Counter_State;
Counters[7].Periodic_Reference_Total := TotalePacchiParziali;
Counters[7].Enable_Reset_Dopo_Salvataggio := TRUE;

// Canale 8 - Totale pacchi settimo codice - parziale
Counters[8].Enable := TRUE;
Counters[8].Nome := CONCAT(STR1:= 'Settimo codice - parziale, VALORE -> ', STR2 := INT_TO_STRING(7));
Counters[8].Enable_Reset_Storico := FALSE;
Counters[8].ResetCounter := DATA_LOGGER.Reset_Operatore;
Counters[8].Daily_Reference_Total := Counters[1].Daily_Counter_State;
Counters[8].Weekly_Reference_Total := Counters[1].Weekly_Counter_State;
Counters[8].Periodic_Reference_Total := TotalePacchiParziali;
Counters[8].Enable_Reset_Dopo_Salvataggio := TRUE;

// Canale 9 - Totale pacchi ottavo codice - parziale
Counters[9].Enable := TRUE;
Counters[9].Nome := CONCAT(STR1:= 'Ottavo codice - parziale, VALORE -> ', STR2 := INT_TO_STRING(8));
Counters[9].Enable_Reset_Storico := FALSE;
Counters[9].ResetCounter := DATA_LOGGER.Reset_Operatore;
Counters[9].Daily_Reference_Total := Counters[1].Daily_Counter_State;
Counters[9].Weekly_Reference_Total := Counters[1].Weekly_Counter_State;
Counters[9].Periodic_Reference_Total := TotalePacchiParziali;
Counters[9].Enable_Reset_Dopo_Salvataggio := TRUE;

// Canale 10 - Totale pacchi nono codice - parziale
Counters[10].Enable := TRUE;
Counters[10].Nome := CONCAT(STR1:= 'Nono codice - parziale, VALORE -> ', STR2 := INT_TO_STRING(9));
Counters[10].Enable_Reset_Storico := FALSE;
Counters[10].ResetCounter := DATA_LOGGER.Reset_Operatore;
Counters[10].Daily_Reference_Total := Counters[1].Daily_Counter_State;
Counters[10].Weekly_Reference_Total := Counters[1].Weekly_Counter_State;
Counters[10].Periodic_Reference_Total := TotalePacchiParziali;
Counters[10].Enable_Reset_Dopo_Salvataggio := TRUE;

// Canale 11 - Totale pacchi decimo codice - parziale
Counters[11].Enable := TRUE;
Counters[11].Nome := CONCAT(STR1:= 'Decimo codice - parziale, VALORE -> ', STR2 := INT_TO_STRING(10));
Counters[11].Enable_Reset_Storico := FALSE;
Counters[11].ResetCounter := DATA_LOGGER.Reset_Operatore;
Counters[11].Daily_Reference_Total := Counters[1].Daily_Counter_State;
Counters[11].Weekly_Reference_Total := Counters[1].Weekly_Counter_State;
Counters[11].Periodic_Reference_Total := TotalePacchiParziali;
Counters[11].Enable_Reset_Dopo_Salvataggio := TRUE;

// Canale 12 - Totale pacchi undicesimo codice - parziale
Counters[12].Enable := TRUE;
Counters[12].Nome := CONCAT(STR1:= 'Undicesimo codice - parziale, VALORE -> ', STR2 := INT_TO_STRING(11));
Counters[12].Enable_Reset_Storico := FALSE;
Counters[12].ResetCounter := DATA_LOGGER.Reset_Operatore;
Counters[12].Daily_Reference_Total := Counters[1].Daily_Counter_State;
Counters[12].Weekly_Reference_Total := Counters[1].Weekly_Counter_State;
Counters[12].Periodic_Reference_Total := TotalePacchiParziali;
Counters[12].Enable_Reset_Dopo_Salvataggio := TRUE;

// Canale 13 - Totale pacchi dodicesimo codice - parziale
Counters[13].Enable := TRUE;
Counters[13].Nome := CONCAT(STR1:= 'Dodicesimo codice - parziale, VALORE -> ', STR2 := INT_TO_STRING(12));
Counters[13].Enable_Reset_Storico := FALSE;
Counters[13].ResetCounter := DATA_LOGGER.Reset_Operatore;
Counters[13].Daily_Reference_Total := Counters[1].Daily_Counter_State;
Counters[13].Weekly_Reference_Total := Counters[1].Weekly_Counter_State;
Counters[13].Periodic_Reference_Total := TotalePacchiParziali;
Counters[13].Enable_Reset_Dopo_Salvataggio := TRUE;

// Canale 14 - Totale pacchi tredicesimo codice - parziale
Counters[14].Enable := TRUE;
Counters[14].Nome := CONCAT(STR1:= 'Tredicesimo codice - parziale, VALORE -> ', STR2 := INT_TO_STRING(13));
Counters[14].Enable_Reset_Storico := FALSE;
Counters[14].ResetCounter := DATA_LOGGER.Reset_Operatore;
Counters[14].Daily_Reference_Total := Counters[1].Daily_Counter_State;
Counters[14].Weekly_Reference_Total := Counters[1].Weekly_Counter_State;
Counters[14].Periodic_Reference_Total := TotalePacchiParziali;
Counters[14].Enable_Reset_Dopo_Salvataggio := TRUE;

// Canale 15 - Totale pacchi quattordicesimo codice - parziale
Counters[15].Enable := TRUE;
Counters[15].Nome := CONCAT(STR1:= 'Quattordicesimo codice - parziale, VALORE -> ', STR2 := INT_TO_STRING(14));
Counters[15].Enable_Reset_Storico := FALSE;
Counters[15].ResetCounter := DATA_LOGGER.Reset_Operatore;
Counters[15].Daily_Reference_Total := Counters[1].Daily_Counter_State;
Counters[15].Weekly_Reference_Total := Counters[1].Weekly_Counter_State;
Counters[15].Periodic_Reference_Total := TotalePacchiParziali;
Counters[15].Enable_Reset_Dopo_Salvataggio := TRUE;

// Canale 16 - Totale pacchi quindicesimo codice - parziale
Counters[16].Enable := TRUE;
Counters[16].Nome := CONCAT(STR1:= 'Quindicesimo codice - parziale, VALORE -> ', STR2 := INT_TO_STRING(15));
Counters[16].Enable_Reset_Storico := FALSE;
Counters[16].ResetCounter := DATA_LOGGER.Reset_Operatore;
Counters[16].Daily_Reference_Total := Counters[1].Daily_Counter_State;
Counters[16].Weekly_Reference_Total := Counters[1].Weekly_Counter_State;
Counters[16].Periodic_Reference_Total := TotalePacchiParziali;
Counters[16].Enable_Reset_Dopo_Salvataggio := TRUE;

(* Reset x evitare false letture *)
PaccoPresoXDataLogger := FALSE;
//DATA_LOGGER.Reset_Operatore := FALSE;
END_ACTION

ACTION _09_CalcolaFormatura:
//Ack 
IF HMI_ErrAckCalcolaFormatura THEN
	HMI_Forming_ErroreCalcoli := 0;
	HMI_ErrAckCalcolaFormatura := FALSE;
	FOR i:= 1 TO MAXFORMING DO
		HMI_Forming_FormaturaAttivata[i] := FALSE;
	END_FOR
END_IF

//Attivazione
FOR i:= 1 TO MAXFORMING DO
	//IF HMI_Forming_Attivazione[i] AND i <=2 AND FALSE THEN
	IF HMI_Forming_Attivazione[i] AND i <=3 AND FALSE THEN
		NCodiciPresenti := 0;
		FOR iform := 1 TO MAXFORMING DO
			FOR icode:=1 TO MAXFORMINGCODE DO
				FOR icode2:=1 TO MAXFORMINGCODE DO
					IF HMI_Forming_CodiciAbilitatiFormatura[i].Code[icode] = Forming[iform].Code[icode] AND Forming[iform].Code[icode] > 0 AND iform <> i THEN
						HMI_Forming_ErroreCalcoli := ErrRipetizioneCodici;		
						HMI_Forming_Attivazione[i] := FALSE; // prueva quitar 
						RETURN;
					END_IF 
				END_FOR
				IF HMI_Forming_CodiciAbilitatiFormatura[i].Code[icode] > 0 THEN
					NCodiciPresenti := NcodiciPresenti+1;
				END_IF
			END_FOR
		END_FOR
		//VErifico che ci sia almento un codice da attivare
		IF NcodiciPresenti = 0 THEN
			HMI_Forming_ErroreCalcoli := ErrNessunCodiciPresente;
			RETURN;
		END_IF
	
		// MEMSET(ADR(Forming[i]),0,SIZEOF(Forming[i])); //prueva Quitar
		IF NOT CalcolaFormaturaTrig AND FALSE  THEN
			HMI_Forming_FormaturaAttivata[i] 	:= FALSE;
			TFCalcoloFormatura.PulisciMemoria 	:= TRUE;
			IF TFCalcoloFormatura.PulisciMemoriaDone THEN	
				HMI_Forming_ErroreCalcoli := 0;
				//Assegno l'ordine tutto a 1 perchè ho solo lastre
				FOR i:= 1 TO MAXFORMINGSLAB DO
					IF i <= HMI_Forming_NumeroElementiDaDepositare THEN
						TFCalcoloFormatura.TipoElementoDep[i] := LASTRA;//Settiamo tutte lastre!!
					ELSE
						TFCalcoloFormatura.TipoElementoDep[i] := TERMINATORE;//Settiamo il resto come terminatore
					END_IF
				END_FOR
				TFCalcoloFormatura.Materiale[e_Tipo_Elemento_Da_Lavorare.LASTRA]		:= HMI_Forming_LastraDaDepositare;
				TFCalcoloFormatura.Materiale[e_Tipo_Elemento_Da_Lavorare.LASTRA].Typology := LASTRA;
				TFCalcoloFormatura.Materiale[e_Tipo_Elemento_Da_Lavorare.FALDA]			:= HMI_Forming_LastraDaDepositare;
				TFCalcoloFormatura.Materiale[e_Tipo_Elemento_Da_Lavorare.FALDA].Typology := FALDA;
				TFCalcoloFormatura.Materiale[e_Tipo_Elemento_Da_Lavorare.QUADROTTA]		:= HMI_Forming_LastraDaDepositare;
				TFCalcoloFormatura.Materiale[e_Tipo_Elemento_Da_Lavorare.QUADROTTA].Typology := QUADROTTA;
				TFCalcoloFormatura.Supporto			:= HMI_Forming_Supporto;	//Assegno la tipologia di supporto
				TFCalcoloFormatura.CalcolaFormatura := TRUE; 		//Lancio esecuzione dei calcoli
				MEMSET(ADR(HMI_Forming_FormaturaCalcolata),0,SIZEOF(HMI_Forming_FormaturaCalcolata));	//Pulisco la memoria di destinazione
				CalcolaFormaturaTrig := TRUE;
				HMI_Forming_Attivazione[i] := FALSE;
				TFCalcoloFormatura.PulisciMemoria := FALSE;
			END_IF
		ELSIF (TFCalcoloFormatura.CalcolaFormaturaDone OR TFCalcoloFormatura.Errore > 0) AND CalcolaFormaturaTrig AND FALSE THEN
			TFCalcoloFormatura.CalcolaFormatura := FALSE;
			IF TFCalcoloFormatura.Errore = 0 THEN
				IDFormatura 			:= IDFormatura+1;
				GUIDFormatura 			:= STRING_TO_UINT(concat(UINT_TO_STRING(NUMERO_MACCHINA),UINT_TO_STRING(IDFormatura)));
				HMI_Forming_GUID 		:= GUIDFormatura;
		
				HMI_Forming_FormaturaCalcolata 	:= TFCalcoloFormatura.FormingSlab;
				MEMSET(ADR(Forming[i]),0,SIZEOF(Forming[i]));	//Pulisco la memoria di destinazione
				Forming[i] 							:= TFCalcoloFormatura.FormingSlab;
				Forming[i].Enable 					:= 1;
				Forming[i].Code 					:= HMI_Forming_CodiciAbilitatiFormatura[i].Code;
				Forming[i].GUID						:= HMI_Forming_GUID;
				Forming[i].Pallet					:= HMI_Forming_Supporto;
				HMI_Forming_IndiceFormaturaAttivata := i;
				HMI_Forming_FormaturaAttivata[i] 	:= TRUE;
			ELSE
				HMI_Forming_ErroreCalcoli := TFCalcoloFormatura.Errore;
			END_IF
			CalcolaFormaturaTrig := FALSE;
			HMI_Forming_Attivazione[i] := FALSE;
		END_IF
	ELSIF HMI_Forming_Attivazione[i] AND FALSE THEN
		memset(destAddr:=ADR(TFCalcoloFormatura.Errore),fillByte:=(UINT_TO_USINT(ErrNumeroMassimoFormatureAmmesse)),n:=SIZEOF(TFCalcoloFormatura.Errore));
	END_IF

	//Disattivazione formatura
	IF HMI_Forming_Disattivazione[i] AND FALSE  THEN
		HMI_Forming_Disattivazione[i] := FALSE;
		MEMSET(ADR(Forming[i]),0,SIZEOF(Forming[i]));	//Pulisco la formatura selezionata e di consegenza la disattivo
	END_IF
		
END_FOR

//IF HMI_Forming_Calcola AND Forming[1].Enable = 1 AND Forming[2].Enable = 1 THEN
//	memset(destAddr:=ADR(TFCalcoloFormatura.Errore),fillByte:=(UINT_TO_USINT(ErrNumeroMassimoFormatureAmmesse)),n:=SIZEOF(TFCalcoloFormatura.Errore));
//	HMI_Forming_Calcola := FALSE;
//Creazione
IF HMI_Forming_Calcola  AND NOT CalcolaFormaturaTrig AND FALSE THEN
	TFCalcoloFormatura.PulisciMemoria := TRUE;
	IF TFCalcoloFormatura.PulisciMemoriaDone THEN	
		HMI_Forming_ErroreCalcoli := 0;
		//Assegno l'ordine tutto a 1 perchè ho solo lastre
		FOR i:= 1 TO MAXFORMINGSLAB DO
			IF i <= HMI_Forming_NumeroElementiDaDepositare THEN
				TFCalcoloFormatura.TipoElementoDep[i] := LASTRA;//Settiamo tutte lastre!!
			ELSE
				TFCalcoloFormatura.TipoElementoDep[i] := TERMINATORE;//Settiamo il resto come terminatore
			END_IF
		END_FOR
		TFCalcoloFormatura.Materiale[e_Tipo_Elemento_Da_Lavorare.LASTRA]		:= HMI_Forming_LastraDaDepositare;
		TFCalcoloFormatura.Materiale[e_Tipo_Elemento_Da_Lavorare.LASTRA].Typology := LASTRA;
		TFCalcoloFormatura.Materiale[e_Tipo_Elemento_Da_Lavorare.FALDA]			:= HMI_Forming_LastraDaDepositare;
		TFCalcoloFormatura.Materiale[e_Tipo_Elemento_Da_Lavorare.FALDA].Typology := FALDA;
		TFCalcoloFormatura.Materiale[e_Tipo_Elemento_Da_Lavorare.QUADROTTA]		:= HMI_Forming_LastraDaDepositare;
		TFCalcoloFormatura.Materiale[e_Tipo_Elemento_Da_Lavorare.QUADROTTA].Typology := QUADROTTA;
		TFCalcoloFormatura.Supporto					:= HMI_Forming_Supporto;	//Assegno la tipologia di supporto
		TFCalcoloFormatura.CalcolaFormatura 		:= HMI_Forming_Calcola; 		//Lancio esecuzione dei calcoli
		TFCalcoloFormatura.NumeroElementiDaDepositare := HMI_Forming_NumeroElementiDaDepositare; 		//Lancio esecuzione dei calcoli
			
		MEMSET(ADR(HMI_Forming_FormaturaCalcolata),0,SIZEOF(HMI_Forming_FormaturaCalcolata));	//Pulisco la memoria di destinazione
		CalcolaFormaturaTrig := TRUE;
		//HMI_Forming_Calcola := FALSE;
		TFCalcoloFormatura.PulisciMemoria := FALSE;
	END_IF

ELSIF HMI_Forming_Calcola AND (TFCalcoloFormatura.CalcolaFormaturaDone OR TFCalcoloFormatura.Errore > 0) AND CalcolaFormaturaTrig AND FALSE THEN
	HMI_Forming_Calcola := FALSE;
	TFCalcoloFormatura.CalcolaFormatura := FALSE;
	IF TFCalcoloFormatura.Errore = 0 THEN
		HMI_Forming_FormaturaCalcolata 	:= TFCalcoloFormatura.FormingSlab;
	//	IDFormatura 			:= IDFormatura+1;
	//	GUIDFormatura 			:= STRING_TO_UINT(concat(UINT_TO_STRING(NUMERO_MACCHINA),UINT_TO_STRING(IDFormatura)));
	//	HMI_Forming_GUID 		:= GUIDFormatura;
		(*FOR i:= 1 TO 2 DO
			IF Forming[i].Enable <> 1 THEN
				MEMSET(ADR(Forming[i]),0,SIZEOF(Forming[i]));	//Pulisco la memoria di destinazione
				HMI_Forming_IndiceFormaturaAttivata := i;
				Forming[i] 			:= TFCalcoloFormatura.FormingSlab;
				Forming[i].Enable 	:= 1;
				Forming[i].Code 	:= HMI_Forming_CodiciAbilitatiFormatura[i].Code;
				Forming[i].GUID		:= HMI_Forming_GUID;
				Forming[i].Pallet	:= HMI_Forming_Supporto;
			ELSE
				CONTINUE;
			END_IF
			EXIT;
		END_FOR*)
		HMI_Forming_FormaturaCreata := TRUE;
	ELSE
		HMI_Forming_ErroreCalcoli := TFCalcoloFormatura.Errore;
	END_IF
	
	CalcolaFormaturaTrig := FALSE;
END_IF
IF FALSE THEN 
	 TFCalcoloFormatura();
END_IF
  

(*//Ack 
IF HMI_ErrAckCalcolaFormatura THEN
	HMI_Forming_ErroreCalcoli := 0;
	HMI_ErrAckCalcolaFormatura := FALSE;
	FOR i:= 1 TO MAXFORMING DO
		HMI_ConfermaAttivazioneFormatura[i] := FALSE;
		HMI_Forming_FormaturaAttivata[i] := FALSE;
	END_FOR
END_IF

//Attivazione
FOR i:= 1 TO MAXFORMING DO
	IF HMI_Forming_Attivazione[i] AND i <=2 THEN
		NCodiciPresenti := 0;
		
		FOR iform := 1 TO MAXFORMING DO
			FOR icode:=1 TO MAXFORMINGCODE DO
				FOR icode2:=1 TO MAXFORMINGCODE DO
					IF HMI_Forming_CodiciAbilitatiFormatura[i].Code[icode] = Forming[iform].Code[icode] AND Forming[iform].Code[icode] > 0 AND iform <> i THEN
						HMI_Forming_ErroreCalcoli := ErrRipetizioneCodici;		
						HMI_Forming_Attivazione[i] := FALSE;
						RETURN;
					END_IF 
				END_FOR
				IF HMI_Forming_CodiciAbilitatiFormatura[i].Code[icode] > 0 THEN
					NCodiciPresenti := NcodiciPresenti+1;
				END_IF
			END_FOR
		END_FOR
		//VErifico che ci sia almento un codice da attivare
		IF NcodiciPresenti = 0 THEN
			HMI_Forming_ErroreCalcoli := ErrNessunCodiciPresente;
			RETURN;
		END_IF
	
		MEMSET(ADR(Forming[i]),0,SIZEOF(Forming[i]));
		IF NOT CalcolaFormaturaTrig  THEN
			HMI_Forming_FormaturaAttivata[i] 	:= FALSE;
			TFCalcoloFormatura.PulisciMemoria 	:= TRUE;
			IF TFCalcoloFormatura.PulisciMemoriaDone THEN	
				HMI_Forming_ErroreCalcoli := 0;
				//Assegno l'ordine tutto a 1 perchè ho solo lastre
				FOR i:= 1 TO MAXFORMINGSLAB DO
					IF i <= HMI_Forming_NumeroElementiDaDepositare THEN
						TFCalcoloFormatura.TipoElementoDep[i] := LASTRA;//Settiamo tutte lastre!!
					ELSE
						TFCalcoloFormatura.TipoElementoDep[i] := TERMINATORE;//Settiamo il resto come terminatore
					END_IF
				END_FOR
				TFCalcoloFormatura.Materiale[e_Tipo_Elemento_Da_Lavorare.LASTRA]		:= HMI_Forming_LastraDaDepositare;
				TFCalcoloFormatura.Materiale[e_Tipo_Elemento_Da_Lavorare.LASTRA].Typology := LASTRA;
				TFCalcoloFormatura.Materiale[e_Tipo_Elemento_Da_Lavorare.FALDA]			:= HMI_Forming_LastraDaDepositare;
				TFCalcoloFormatura.Materiale[e_Tipo_Elemento_Da_Lavorare.FALDA].Typology := FALDA;
				TFCalcoloFormatura.Materiale[e_Tipo_Elemento_Da_Lavorare.QUADROTTA]		:= HMI_Forming_LastraDaDepositare;
				TFCalcoloFormatura.Materiale[e_Tipo_Elemento_Da_Lavorare.QUADROTTA].Typology := QUADROTTA;
				TFCalcoloFormatura.Supporto			:= HMI_Forming_Supporto;	//Assegno la tipologia di supporto
				TFCalcoloFormatura.CalcolaFormatura := TRUE; 		//Lancio esecuzione dei calcoli
				MEMSET(ADR(HMI_Forming_FormaturaCalcolata),0,SIZEOF(HMI_Forming_FormaturaCalcolata));	//Pulisco la memoria di destinazione
				HMI_Forming_Attivazione[i] := FALSE;
				TFCalcoloFormatura.PulisciMemoria := FALSE;
				CalcolaFormaturaTrig := TRUE;
			END_IF
		ELSIF (TFCalcoloFormatura.CalcolaFormaturaDone OR TFCalcoloFormatura.Errore > 0) AND CalcolaFormaturaTrig THEN
			//CalcolaFormaturaTrig := FALSE;
			TFCalcoloFormatura.CalcolaFormatura := FALSE;
			IF TFCalcoloFormatura.Errore = 0 THEN
				IDFormatura 			:= IDFormatura+1;
				GUIDFormatura 			:= STRING_TO_UINT(concat(UINT_TO_STRING(NUMERO_MACCHINA),UINT_TO_STRING(IDFormatura)));
				HMI_Forming_GUID 		:= GUIDFormatura;
		
				HMI_Forming_FormaturaCalcolata 	:= TFCalcoloFormatura.FormingSlab;
				MEMSET(ADR(Forming[i]),0,SIZEOF(Forming[i]));	//Pulisco la memoria di destinazione
				Forming[i] 							:= TFCalcoloFormatura.FormingSlab;
				Forming[i].Enable 					:= 1;
				Forming[i].Code 					:= HMI_Forming_CodiciAbilitatiFormatura[i].Code;
				Forming[i].GUID						:= HMI_Forming_GUID;
				Forming[i].Pallet					:= HMI_Forming_Supporto;
				HMI_Forming_IndiceFormaturaAttivata := i;
				HMI_Forming_FormaturaAttivata[i] 	:= TRUE;
			ELSE
				HMI_Forming_ErroreCalcoli := TFCalcoloFormatura.Errore;
			END_IF
			HMI_Forming_Attivazione[i] := FALSE;
		END_IF
	ELSIF HMI_Forming_Attivazione[i] THEN
		memset(destAddr:=ADR(TFCalcoloFormatura.Errore),fillByte:=(UINT_TO_USINT(ErrNumeroMassimoFormatureAmmesse)),n:=SIZEOF(TFCalcoloFormatura.Errore));
	END_IF

	//Disattivazione formatura
	IF HMI_Forming_Disattivazione[i] THEN
		HMI_Forming_Disattivazione[i] := FALSE;
		MEMSET(ADR(Forming[i]),0,SIZEOF(Forming[i]));	//Pulisco la formatura selezionata e di consegenza la disattivo
	END_IF
		
END_FOR

//IF HMI_Forming_Calcola AND Forming[1].Enable = 1 AND Forming[2].Enable = 1 THEN
//	memset(destAddr:=ADR(TFCalcoloFormatura.Errore),fillByte:=(UINT_TO_USINT(ErrNumeroMassimoFormatureAmmesse)),n:=SIZEOF(TFCalcoloFormatura.Errore));
//	HMI_Forming_Calcola := FALSE;
//Creazione
IF HMI_Forming_Calcola  AND NOT CalcolaFormaturaTrig  THEN
	TFCalcoloFormatura.PulisciMemoria := TRUE;
	IF TFCalcoloFormatura.PulisciMemoriaDone THEN	
		TFCalcoloFormatura.PulisciMemoria := FALSE;
		HMI_Forming_ErroreCalcoli := 0;
		CalcolaFormaturaTrig := TRUE;
		//Assegno l'ordine tutto a 1 perchè ho solo lastre
		FOR i:= 1 TO MAXFORMINGSLAB DO
			IF i <= HMI_Forming_NumeroElementiDaDepositare THEN
				TFCalcoloFormatura.TipoElementoDep[i] := LASTRA;//Settiamo tutte lastre!!
			ELSE
				TFCalcoloFormatura.TipoElementoDep[i] := TERMINATORE;//Settiamo il resto come terminatore
			END_IF
		END_FOR
		TFCalcoloFormatura.Materiale[e_Tipo_Elemento_Da_Lavorare.LASTRA]		:= HMI_Forming_LastraDaDepositare;
		TFCalcoloFormatura.Materiale[e_Tipo_Elemento_Da_Lavorare.LASTRA].Typology := LASTRA;
		TFCalcoloFormatura.Materiale[e_Tipo_Elemento_Da_Lavorare.FALDA]			:= HMI_Forming_LastraDaDepositare;
		TFCalcoloFormatura.Materiale[e_Tipo_Elemento_Da_Lavorare.FALDA].Typology := FALDA;
		TFCalcoloFormatura.Materiale[e_Tipo_Elemento_Da_Lavorare.QUADROTTA]		:= HMI_Forming_LastraDaDepositare;
		TFCalcoloFormatura.Materiale[e_Tipo_Elemento_Da_Lavorare.QUADROTTA].Typology := QUADROTTA;
		TFCalcoloFormatura.Supporto					:= HMI_Forming_Supporto;	//Assegno la tipologia di supporto
		TFCalcoloFormatura.CalcolaFormatura 		:= HMI_Forming_Calcola; 		//Lancio esecuzione dei calcoli
		TFCalcoloFormatura.NumeroElementiDaDepositare := HMI_Forming_NumeroElementiDaDepositare; 		//Lancio esecuzione dei calcoli
			
		MEMSET(ADR(HMI_Forming_FormaturaCalcolata),0,SIZEOF(HMI_Forming_FormaturaCalcolata));	//Pulisco la memoria di destinazione
		//HMI_Forming_Calcola := FALSE;
	END_IF

ELSIF HMI_Forming_Calcola AND (TFCalcoloFormatura.CalcolaFormaturaDone OR TFCalcoloFormatura.Errore > 0) AND CalcolaFormaturaTrig THEN
	HMI_Forming_Calcola := FALSE;
	TFCalcoloFormatura.CalcolaFormatura := FALSE;
	IF TFCalcoloFormatura.Errore = 0 THEN
		HMI_Forming_FormaturaCalcolata 	:= TFCalcoloFormatura.FormingSlab;
	//	IDFormatura 			:= IDFormatura+1;
	//	GUIDFormatura 			:= STRING_TO_UINT(concat(UINT_TO_STRING(NUMERO_MACCHINA),UINT_TO_STRING(IDFormatura)));
	//	HMI_Forming_GUID 		:= GUIDFormatura;
		(*FOR i:= 1 TO 2 DO
			IF Forming[i].Enable <> 1 THEN
				MEMSET(ADR(Forming[i]),0,SIZEOF(Forming[i]));	//Pulisco la memoria di destinazione
				HMI_Forming_IndiceFormaturaAttivata := i;
				Forming[i] 			:= TFCalcoloFormatura.FormingSlab;
				Forming[i].Enable 	:= 1;
				Forming[i].Code 	:= HMI_Forming_CodiciAbilitatiFormatura[i].Code;
				Forming[i].GUID		:= HMI_Forming_GUID;
				Forming[i].Pallet	:= HMI_Forming_Supporto;
			ELSE
				CONTINUE;
			END_IF
			EXIT;
		END_FOR*)
		HMI_Forming_FormaturaCreata := TRUE;
	ELSE
		HMI_Forming_ErroreCalcoli := TFCalcoloFormatura.Errore;
	END_IF
	
	CalcolaFormaturaTrig := FALSE;
END_IF

TFCalcoloFormatura();*)
END_ACTION

ACTION _10_PackModifier:
//Filtro le FTC delle postazioni
FOR i := 1 TO MAXAREAPRESENT DO
	FiltroFTCPalletPerManuale[i].FilterTime_OFF := 3000;
	FiltroFTCPalletPerManuale[i].FilterTime_ON 	:= 3000;
	FiltroFTCPalletPerManuale[i].IN_Signal 		:= I_PHPresenzaPallet[i];
	FiltroFTCPalletPerManuale[i]();
END_FOR

IF MachinePalletizer_TF.CmdExe.Code = CmdNOP THEN
	FOR i:= 1 TO MAXAREAPRESENT DO
		IF HMI_NumeroPezziPresentiPostazione[i] <> WorkAreaState[i].P-1 THEN
			WorkAreaState[i].P := HMI_NumeroPezziPresentiPostazione[i]+1;
		END_IF	
		
		IF WorkAreaState[i].PackPointerModified THEN//Se sto facendo una modifica da HMI
			WorkAreaState[i].PackPointer:= MIN(MAX(1,WorkAreaState[i].PackPointer ),MAXFORMINGSLAB);//limito i valori con quelli ammissibili
			IF WorkAreaState[i].PackPointer > WorkAreaState[i].P THEN 
				IF (WorkAreaState[i].PackPointer - WorkAreaState[i].P) = 1 THEN
					WorkAreaState[i].P := WorkAreaState[i].P+1;
				ELSE 
					WorkAreaState[i].P := WorkAreaState[i].PackPointer+1;	
				END_IF
			ELSE
				IF (WorkAreaState[i].PackPointer - WorkAreaState[i].P) = -1 THEN
					WorkAreaState[i].P := WorkAreaState[i].P-1;
				ELSE 
					WorkAreaState[i].P := WorkAreaState[i].PackPointer+1;	
				END_IF
			END_IF
			WorkAreaState[i].Slow := 1;
			WorkAreaState[i].PackPointerModified := FALSE;
			WorkAreaState[i].PackPointer := -1;
		END_IF
		//
		HMI_NumeroPezziPresentiPostazione[i] := MAX(0,WorkAreaState[i].P-1);
		
		AggiuntaPalletManuale(WorkArea := ADR(WorkArea),
									WorkAreaState := ADR(WorkAreaState),
									WorkAreaNumber := i,
									Forming := ADR(Forming),
									Pallet := ADR(Pallet),
									Layer := ADR(Layer),
									ProgressiveNrWA := ADR(ProgressiveNrWA),
									CodicePostazione := WorkAreaState[i].Code,
									AbilitaAssegnazioneCodicePiazzoleConPaccoSuRibaltino := TRUE,
									PH_Presenza := FiltroFTCPalletPerManuale[i].Out_Signal_Filtrato);	
	END_FOR
END_IF
END_ACTION

ACTION _11_CalcolaListaProduzione:
{region "Gestione zona GLOBALE - Postazioni da 1 a 8"}


//#############################################################################################################

{region "Gestione zona GLOBALE - Postazioni da 1 a 8"}

//Traferisco i valori dei supporti della lista 1 nella lista 2 e 3
RequestPickingListFromHMI[2].SupportPianoFerro 	:= RequestPickingListFromHMI[1].SupportPianoFerro;		  
RequestPickingListFromHMI[3].SupportPianoFerro 	:= RequestPickingListFromHMI[1].SupportPianoFerro;		  
RequestPickingListFromHMI[2].SupportPianoLegno 	:= RequestPickingListFromHMI[1].SupportPianoLegno;		  
RequestPickingListFromHMI[3].SupportPianoLegno 	:= RequestPickingListFromHMI[1].SupportPianoLegno;		  
RequestPickingListFromHMI[2].SupportVertBundle 	:= RequestPickingListFromHMI[1].SupportVertBundle;		  
RequestPickingListFromHMI[3].SupportVertBundle 	:= RequestPickingListFromHMI[1].SupportVertBundle;		  
RequestPickingListFromHMI[2].SupportVertCav 	:= RequestPickingListFromHMI[1].SupportVertCav;		  
RequestPickingListFromHMI[3].SupportVertCav 	:= RequestPickingListFromHMI[1].SupportVertCav;		  
RequestPickingListFromHMI[2].SupportVertCav 	:= RequestPickingListFromHMI[1].SupportVertCav;		  
RequestPickingListFromHMI[3].SupportVertCav 	:= RequestPickingListFromHMI[1].SupportVertCav;		  

FOR LoopLista := 1 TO 3 DO
	IdxLista := LoopLista;		 
	 // IdxLista := 2;		  
	CASE IdxLista OF	 
		1: Iforstart := 1; Iforend := MAXAREAPRESENT;
		2: Iforstart := 1; Iforend := 4;
		3: Iforstart := 5; Iforend := MAXAREAPRESENT;
	END_CASE	 
	IF MachinePalletizer_TF.IN.Mode.Man AND
		(MachinePalletizer_TF.CmdExe.Code = CmdNOP OR MachinePalletizer_TF.CmdExe.Code = CmdMAN) THEN

//--------------------------------------------------------
			//AZZERAMENTO (Reset) lista di picking	
//--------------------------------------------------------		 
			IF Cmd_AzzeraLista[IdxLista] THEN
				IF Prueva THEN
					MissionClr := ADR(Mission) ;
	 				MEMSET(destAddr := ADR(MissionClr^),fillByte := 0 , n := SIZEOF(MissionClr^));
				END_IF
					ClrEstructura := ADR(PosCavalleteOrdenPikin) ;
					MEMSET(destAddr := ADR(ClrEstructura^),fillByte := 0 , n := SIZEOF(ClrEstructura^));	  
					NuEstacionesPiking := 0 ;	  
					NuEstacionPiking   := 0 ;
					NuPosGuiroPiking := 0;
					PosFinOrdenPikingCaballete := 0 ;
					
					MultiplesCavalletesReceta := FALSE ;
					CoordenadaPasillo0_Y := 0 ;
					CoordenadaPasillo180_Y := 0 ;
				
				//FOR i:= 1 TO 3 DO
						//CalcolaFormingRT2[i] := FALSE ;
					CalcolaFormingRT[IdxLista] := FALSE ;
					CalcolaFormingRT2[IdxLista] := FALSE ;	 
						//#Añadido 4_7_2025########################
					Formacion_bandelCalOk[IdxLista]			:= FALSE ;
					Formacion_FrameCalOk[IdxLista]			:= FALSE ;
					Formacion_De_listaOk[IdxLista]			:= FALSE ;
					FormaturaAFRAMERT[IdxLista]		   	:=	FormingEmpty;
					FormaturaBundleRT[IdxLista]	 		:=	FormingEmpty;
				//Añadido 4_7_2025##########################
						
				// END_FOR
				ActualPickingListFromHMI[IdxLista].State := e_StatoWorkOrder.NON_ESEGUITO;
				HMI_NumeroLastreDepOrdineAttuale[IdxLista] := 0; 
				//Disattivazione formatura
				Forming[1] := FormingEmpty;	//Pulisco la formatura selezionata e di consegenza la disattivo
				Forming[2] := FormingEmpty;	//Pulisco la formatura selezionata e di consegenza la disattivo
				Forming[3] := FormingEmpty;	//Pulisco la formatura selezionata e di consegenza la disattivo
				Forming[4] := FormingEmpty;	//Pulisco la formatura selezionata e di consegenza la disattivo
				ActualPickingListFromHMI[IdxLista].State := e_StatoWorkOrder.NON_ESEGUITO;
				Cmd_AttivaLista[IdxLista] := FALSE;
				HMI_Forming_NumeroElementiDaDepositare := 0;
 				RequestPickingListFromHMI[IdxLista].SlabNumber :=0;
	 
				//Azzero le liste per le postazioni dove non avviene la pallettizzazione
				FOR i:= Iforstart TO Iforend DO	
					TFClearWorkAreaArray(ADR(Workarea),ADR(WorkAreaState),k:=i);
					HMI_WorkAreaDataPicking[i].Destinazione := FALSE;
					HMI_WorkAreaDataPicking[i].NumElementiDaLavorare := 0;
					WorkAreaState[i].P 			:= 1;
					WorkAreaProductionList[i] 	:= ListaEmpty;
					WorkAreaOffset[i].Y 		:= 0;
					//HMI_NumeroPezziPresentiPostazione[i] 	:= 0; // Quitado Para No resetear posiciones
					NumeroPezziPresentiPostazioneStart[i] 	:= 0;
					WorkAreaProductionList[i].Stato 		:= e_Stato_ListaDiProduzione.LISTA_PROD_ASSENTE;	 
				END_FOR			  
				ActualPickingListFromHMI[IdxLista].SlabNumber 		  			:= 0;
				ActualPickingListFromHMI[IdxLista].SlabDimension.XDim 			:= 0;
				ActualPickingListFromHMI[IdxLista].SlabDimension.YDim 			:= 0;
				ActualPickingListFromHMI[IdxLista].SlabDimension.ZDim 			:= 0;
				ActualPickingListFromHMI[IdxLista].SupportPianoLegno 			:= SupportDataEmpty;
				ActualPickingListFromHMI[IdxLista].SupportPianoFerro 			:= SupportDataEmpty;
				ActualPickingListFromHMI[IdxLista].SupportVertBundle 			:= SupportDataEmpty;
				ActualPickingListFromHMI[IdxLista].SupportVertCav 			 	:= SupportDataEmpty;
				
				HMI_ErroreCalcoloLista 		:= 0;
				Cmd_CalcolaLista[IdxLista] 	:= FALSE;
				HMI_Forming_Attivazione[IdxLista] 	:= FALSE;//attivo nuova formatura
				Cmd_AzzeraLista[IdxLista] := FALSE;
				//Ack 
				//IF HMI_ErrAckCalcolaFormatura THEN
					HMI_Forming_ErroreCalcoli := 0;
					HMI_ErrAckCalcolaFormatura := FALSE;
					FOR i:= 1 TO MAXFORMING DO
						HMI_ConfermaAttivazioneFormatura[i] := FALSE;
						HMI_Forming_FormaturaAttivata[i] := FALSE;
					END_FOR
				//END_IF
				CalcolaFormaturaTrig := FALSE;
			END_IF



//--------------------------------------------------------
		// COMANDO ATTIVAZIONE  lista di picking	
//--------------------------------------------------------		 		  
			//Se non ho una Destinazione impostata, Num.pezzi impostato, o Num.pezzi richiesto...
			//	Resetto il comando		
					IF Cmd_AttivaLista[1] = TRUE  THEN
						IF 	(HMI_WorkAreaDataPicking[1].Destinazione =0 AND 
							HMI_WorkAreaDataPicking[2].Destinazione =0 AND
							HMI_WorkAreaDataPicking[3].Destinazione =0 AND 
							HMI_WorkAreaDataPicking[4].Destinazione =0 AND	 
							HMI_WorkAreaDataPicking[5].Destinazione =0 AND 
							HMI_WorkAreaDataPicking[6].Destinazione =0 AND
							HMI_WorkAreaDataPicking[7].Destinazione =0 AND 
							HMI_WorkAreaDataPicking[8].Destinazione =0)							 
							OR
							(HMI_NumeroPezziPresentiPostazione[1] =0 AND 
							HMI_NumeroPezziPresentiPostazione[2] =0 AND
							HMI_NumeroPezziPresentiPostazione[3] =0 AND 
							HMI_NumeroPezziPresentiPostazione[4] =0 AND
							HMI_NumeroPezziPresentiPostazione[5] =0 AND 
	 						HMI_NumeroPezziPresentiPostazione[6] =0 AND
							HMI_NumeroPezziPresentiPostazione[7] =0 AND 
							HMI_NumeroPezziPresentiPostazione[8] =0)
							OR	 	 
							RequestPickingListFromHMI[1].SlabNumber = 0	 
						THEN
							Cmd_AttivaLista[1] := FALSE;
						 END_IF
					END_IF		  
					IF Cmd_AttivaLista[2] = TRUE  THEN
						IF 	(HMI_WorkAreaDataPicking[1].Destinazione =0 AND 
							HMI_WorkAreaDataPicking[2].Destinazione =0 AND
							HMI_WorkAreaDataPicking[3].Destinazione =0 AND 
							HMI_WorkAreaDataPicking[4].Destinazione =0)
							OR
							(HMI_NumeroPezziPresentiPostazione[1] =0 AND 
							HMI_NumeroPezziPresentiPostazione[2] =0 AND
							HMI_NumeroPezziPresentiPostazione[3] =0 AND 
							HMI_NumeroPezziPresentiPostazione[4] =0)
							OR	 
							RequestPickingListFromHMI[2].SlabNumber = 0	 	 
						THEN
							Cmd_AttivaLista[2] := FALSE;
						 END_IF
					END_IF		
					IF Cmd_AttivaLista[3] = TRUE  THEN
						IF 	(HMI_WorkAreaDataPicking[5].Destinazione =0 AND 
							HMI_WorkAreaDataPicking[6].Destinazione =0 AND
							HMI_WorkAreaDataPicking[7].Destinazione =0 AND 
							HMI_WorkAreaDataPicking[8].Destinazione =0)
							OR
							(HMI_NumeroPezziPresentiPostazione[5] =0 AND 
							HMI_NumeroPezziPresentiPostazione[6] =0 AND
							HMI_NumeroPezziPresentiPostazione[7] =0 AND 
							HMI_NumeroPezziPresentiPostazione[8] =0)
							OR	 	 
							RequestPickingListFromHMI[3].SlabNumber = 0	 	 
						THEN
							Cmd_AttivaLista[3] := FALSE;
						 END_IF
					END_IF		
{Region "Prmer Bucle cuenta las piezas a coger y rellena el workareastate Con el Tipo Palet"}

			// COMANDO ATTIVAZIONE  lista di picking	
		    IF Cmd_AttivaLista[IdxLista] AND ActualPickingListFromHMI[IdxLista].State <> e_StatoWorkOrder.IN_ESECUZIONE THEN
				ElementiDaDepositare[IdxLista]   :=0;
				HMI_ErroreCalcoloLista := 0;
				HMI_NumeroLastreDepOrdineAttuale[IdxLista] := 0;
				FOR i:= Iforstart TO Iforend DO	
					//HMI_WorkAreaDataPicking[i].Destinazione := FALSE;
					//HMI_WorkAreaDataPicking[i].NumElementiDaLavorare := 0;
					WorkAreaState[i].P := 1;
					WorkAreaProductionList[i] := ListaEmpty;
				END_FOR	 
				
				FOR i:= Iforstart TO Iforend DO	
					IF NOT HMI_WorkAreaDataPicking[i].Destinazione THEN
						ElementiDaDepositare[IdxLista] := ElementiDaDepositare[IdxLista] +HMI_WorkAreaDataPicking[i].NumElementiDaLavorare;
						WorkAreaState[i].P := HMI_WorkAreaDataPicking[i].NumElementiDaLavorare +1;
						CASE HMI_WorkAreaDataPicking[i].Typology OF
							LEGNO_PIANO,TELAIO_PIANO:
								WorkareaState[i].Supporto.Tipologia := e_Tipo_Pallet.CASSA_STANDARD;
							A_FRAME_VERT:	
								WorkareaState[i].Supporto.Tipologia := e_Tipo_Pallet.CAVALLETTO;
								
							IF HMI_WorkAreaDataPicking[i].NumElementiDaLavorare > 0 THEN 
								NuEstacionesPiking := NuEstacionesPiking + 1 ;	
								PosCavalleteOrdenPikin[i]	:=  e_Tipo_Pallet.CAVALLETTO;  
							END_IF
							BUNDLE_VERT:
								WorkareaState[i].Supporto.Tipologia := e_Tipo_Pallet.BUNDLE;	
							
						 ELSE
								WorkareaState[i].Supporto.Tipologia := e_Tipo_Pallet.CASSA_STANDARD;		   
						 END_CASE
					ELSE
						NumPostazioneDeposito := i; NuEstacionPiking := i;
						
						HMI_WorkAreaDataPicking[NumPostazioneDeposito].NumElementiDaLavorare := RequestPickingListFromHMI[IdxLista].SlabNumber;
						CASE HMI_WorkAreaDataPicking[i].Typology OF
							LEGNO_PIANO,TELAIO_PIANO:
								WorkareaState[i].Supporto.Tipologia := e_Tipo_Pallet.CASSA_STANDARD;
							A_FRAME_VERT:	
								WorkareaState[i].Supporto.Tipologia := e_Tipo_Pallet.CAVALLETTO;
								NuEstacionesPiking := NuEstacionesPiking + 1 ;	
								PosCavalleteOrdenPikin[i]	:=  e_Tipo_Pallet.CAVALLETTO;  	 
							BUNDLE_VERT:
								WorkareaState[i].Supporto.Tipologia := e_Tipo_Pallet.BUNDLE;	
								
							
						 ELSE
								WorkareaState[i].Supporto.Tipologia := e_Tipo_Pallet.CASSA_STANDARD;		   
						 END_CASE
					END_IF

		  
//HMI_NumeroPezziPresentiPostazione[i] := WorkAreaState[i].P -1; //NB:cancellato xckè alla attivazione azzerava il num.pezzi presenti sulle postazioni di prelievo
				END_FOR
	
				IF ElementiDaDepositare[IdxLista] <= HMI_WorkAreaDataPicking[NumPostazioneDeposito].NumElementiDaLavorare THEN
					ActualPickingListFromHMI[IdxLista] 		:= RequestPickingListFromHMI[IdxLista];
					ActualPickingListFromHMI[IdxLista].State 	:= e_StatoWorkOrder.DA_ESEGUIRE;

				ELSE
					HMI_ErroreCalcoloLista := 1;
				END_IF
				Cmd_AttivaLista[IdxLista] 				:= FALSE;
				 
			ELSE
				Cmd_AttivaLista[IdxLista] 				:= FALSE;
				 
			END_IF
{endregion}	

{region "Cotas posicione de trabajo"}

//--------------------------------------------------------------------				
//////// attivazione lista di picking : StatoWorkOrder.DA_ESEGUIRE ///
//--------------------------------------------------------------------				
			IF ActualPickingListFromHMI[IdxLista].State = e_StatoWorkOrder.DA_ESEGUIRE  THEN
				ListaInEsecuzione[IdxLista] := FALSE;
				NumeroListaInEsecuzione := 0;
			
				(* Inserimento sequenza di prelievo dalle postazioni in base al quello che l'operatore ha editato da HMI*)
				ElementiDaDepositare[IdxLista] := 0;
				ElementiElaborati[IdxLista]    := 1;
				NumPostazioneDeposito := 0;
				//FOR i:= 1 TO MAXAREAPRESENT DO
				//	WorkAreaState[i].P := 1;
				//END_FOR		
				
				FOR i:= Iforstart TO Iforend DO//---------- For 1 HMI_WorkAreaDataPicking[i].Destinazione 
					IF HMI_WorkAreaDataPicking[i].Destinazione THEN  //-------> Palet destino
						NumPostazioneDeposito := i;
						HMI_WorkAreaDataPicking[NumPostazioneDeposito].NumElementiDaLavorare 	:= RequestPickingListFromHMI[IdxLista].SlabNumber;
						(*CASE HMI_WorkAreaDataPicking[i].Typology OF     // case Pricipal1*)		 
						CASE HMI_WorkAreaDataPicking[NumPostazioneDeposito].Typology OF     // case Pricipal1	
							(* Se ho un legno in piano *)	 
							LEGNO_PIANO:	
								WorkAreaState[NumPostazioneDeposito].Supporto.Code 						:= ActualPickingListFromHMI[IdxLista].SupportPianoLegno.Code;
								WorkAreaState[NumPostazioneDeposito].Supporto.AltezzaDenteRitenuta 		:= ActualPickingListFromHMI[IdxLista].SupportPianoLegno.DimBaseUtile;
								WorkAreaState[NumPostazioneDeposito].Supporto.DimVertice 				:= ActualPickingListFromHMI[IdxLista].SupportPianoLegno.DimVertice;
								WorkAreaState[NumPostazioneDeposito].Supporto.HMAX 						:= ActualPickingListFromHMI[IdxLista].SupportPianoLegno.HMAX;
								WorkAreaState[NumPostazioneDeposito].Supporto.Tipologia 				:= e_Tipo_Pallet.CASSA_STANDARD;//ActualPickingListFromHMI.Support.Tipologia;
								WorkAreaState[NumPostazioneDeposito].Supporto.XDim 						:= ActualPickingListFromHMI[IdxLista].SupportPianoLegno.XDim;
								WorkAreaState[NumPostazioneDeposito].Supporto.YDim 						:= ActualPickingListFromHMI[IdxLista].SupportPianoLegno.YDim;
								WorkAreaState[NumPostazioneDeposito].Supporto.ZDim 						:= ActualPickingListFromHMI[IdxLista].SupportPianoLegno.ZDim;
								WorkAreaOffset[NumPostazioneDeposito].Y 								:= OFFSET_POSTAZIONE_LEGNO + ActualPickingListFromHMI[IdxLista].SupportPianoLegno.YDim/2;//ATTENZIONE!!! per poter lavorare in centro con i supporti pari, questa misura è la distanza tra il riscontro bundle verticale e il centro postazione PARI
								
								CASE HMI_WorkAreaDataPicking[NumPostazioneDeposito].Typology OF
									LEGNO_PIANO:
										 		WorkAreaProductionList[NumPostazioneDeposito].Support := WorkAreaState[NumPostazioneDeposito].Supporto;
												WorkAreaProductionList[NumPostazioneDeposito].Support.Tipologia	:= e_Tipo_Pallet.CASSA_STANDARD; 
									TELAIO_PIANO:
										 		WorkAreaProductionList[NumPostazioneDeposito].Support := WorkAreaState[NumPostazioneDeposito].Supporto;
												WorkAreaProductionList[NumPostazioneDeposito].Support.Tipologia	:= e_Tipo_Pallet.CASSA_STANDARD; 
									BUNDLE_VERT:
										 		WorkAreaProductionList[NumPostazioneDeposito].Support := WorkAreaState[NumPostazioneDeposito].Supporto;
												WorkAreaProductionList[NumPostazioneDeposito].Support.Tipologia	:= e_Tipo_Pallet.BUNDLE; 
												
									A_FRAME_VERT:
										 		WorkAreaProductionList[NumPostazioneDeposito].Support := WorkAreaState[NumPostazioneDeposito].Supporto;
												WorkAreaProductionList[NumPostazioneDeposito].Support.Tipologia	:= e_Tipo_Pallet.CAVALLETTO; 
												
								END_CASE
								FOR j:= Iforstart TO Iforend DO
									IF NOT HMI_WorkAreaDataPicking[j].Destinazione THEN
										IF HMI_WorkAreaDataPicking[j].NumElementiDaLavorare >= 1 THEN
											ElementiDaDepositare[IdxLista] := ElementiElaborati[IdxLista] + HMI_WorkAreaDataPicking[j].NumElementiDaLavorare;
											FOR k := ElementiElaborati[IdxLista] TO ElementiDaDepositare[IdxLista]-1 DO	
												WorkAreaProductionList[NumPostazioneDeposito].PElementList[k].WA_PRELIEVO := j;
												WorkAreaProductionList[NumPostazioneDeposito].PElementList[k].WA_DEPOSITO := i;	
												ElementiElaborati[IdxLista] := ElementiElaborati[IdxLista]+1; 
											END_FOR
											CASE HMI_WorkAreaDataPicking[j].Typology OF 
												(* Se ho una cassa pianale in legno *)
												LEGNO_PIANO:
													WorkAreaState[j].Supporto.Code 					:= ActualPickingListFromHMI[IdxLista].SupportPianoLegno.Code;
													WorkAreaState[j].Supporto.DimBaseUtile		 	:= ActualPickingListFromHMI[IdxLista].SupportPianoLegno.DimBaseUtile;
													WorkAreaState[j].Supporto.AltezzaDenteRitenuta 	:= ActualPickingListFromHMI[IdxLista].SupportPianoLegno.ZDim+20;
													WorkAreaState[j].Supporto.DimVertice 			:= ActualPickingListFromHMI[IdxLista].SupportPianoLegno.DimVertice;
													WorkAreaState[j].Supporto.HMAX 					:= ActualPickingListFromHMI[IdxLista].SupportPianoLegno.HMAX;
													WorkAreaState[j].Supporto.Tipologia 			:= e_Tipo_Pallet.CASSA_STANDARD;//ActualPickingListFromHMI[1].Support.Tipologia;
													WorkAreaState[j].Supporto.XDim 					:= ActualPickingListFromHMI[IdxLista].SupportPianoLegno.XDim;
													WorkAreaState[j].Supporto.YDim 					:= ActualPickingListFromHMI[IdxLista].SupportPianoLegno.YDim;
													WorkAreaState[j].Supporto.ZDim 					:= ActualPickingListFromHMI[IdxLista].SupportPianoLegno.ZDim;
													WorkAreaOffset[j].Y 							:= OFFSET_POSTAZIONE_LEGNO + ActualPickingListFromHMI[IdxLista].SupportPianoLegno.YDim/2;//ATTENZIONE!!! per poter lavorare in centro con i supporti pari, questa misura è la distanza tra il riscontro bundle verticale e il centro postazione PARI
												(* Se ho una cassa pianale in ferro su supporto *)
												TELAIO_PIANO:
													WorkAreaState[j].Supporto.Code 					:= ActualPickingListFromHMI[IdxLista].SupportPianoFerro.Code;
													WorkAreaState[j].Supporto.DimBaseUtile		 	:= ActualPickingListFromHMI[IdxLista].SupportPianoFerro.DimBaseUtile;
													WorkAreaState[j].Supporto.AltezzaDenteRitenuta 	:= ActualPickingListFromHMI[IdxLista].SupportPianoFerro.ZDim+20;
													WorkAreaState[j].Supporto.DimVertice 			:= ActualPickingListFromHMI[IdxLista].SupportPianoFerro.DimVertice;
													WorkAreaState[j].Supporto.HMAX 					:= ActualPickingListFromHMI[IdxLista].SupportPianoFerro.HMAX;
													WorkAreaState[j].Supporto.Tipologia 			:=  e_Tipo_Pallet.CASSA_STANDARD;//ActualPickingListFromHMI[1].Support.Tipologia;
													WorkAreaState[j].Supporto.XDim 					:= ActualPickingListFromHMI[IdxLista].SupportPianoFerro.XDim;
													WorkAreaState[j].Supporto.YDim 					:= ActualPickingListFromHMI[IdxLista].SupportPianoFerro.YDim;
													WorkAreaState[j].Supporto.ZDim 					:= ActualPickingListFromHMI[IdxLista].SupportPianoFerro.ZDim;
													WorkAreaOffset[j].Y 							:= OFFSET_POSTAZIONE_TELAIO - ActualPickingListFromHMI[IdxLista].SupportPianoFerro.YDim/2;//ATTENZIONE!!! per poter lavorare in centro con i supporti pari, questa misura è la distanza tra il riscontro bundle verticale e il centro postazione PARI
												(* Se ho un bundle *)
												BUNDLE_VERT:
													//WorkAreaState[j].P := ElementiDaDepositare;
													WorkAreaState[j].Supporto.Code 					:= ActualPickingListFromHMI[IdxLista].SupportVertBundle.Code;
													WorkAreaState[j].Supporto.DimBaseUtile		 	:= ActualPickingListFromHMI[IdxLista].SupportVertBundle.DimBaseUtile;
													WorkAreaState[j].Supporto.AltezzaDenteRitenuta 	:= ActualPickingListFromHMI[IdxLista].SupportVertBundle.ZDim+20;
													WorkAreaState[j].Supporto.DimVertice 			:= ActualPickingListFromHMI[IdxLista].SupportVertBundle.DimVertice;
													WorkAreaState[j].Supporto.HMAX 					:= ActualPickingListFromHMI[IdxLista].SupportVertBundle.HMAX;
													WorkAreaState[j].Supporto.Tipologia 			:= e_Tipo_Pallet.BUNDLE;//ActualPickingListFromHMI.SupportVert.Tipologia;
													WorkAreaState[j].Supporto.XDim 					:= ActualPickingListFromHMI[IdxLista].SupportVertBundle.XDim;
													WorkAreaState[j].Supporto.YDim 					:= ActualPickingListFromHMI[IdxLista].SupportVertBundle.YDim;
													WorkAreaState[j].Supporto.ZDim 					:= ActualPickingListFromHMI[IdxLista].SupportVertBundle.ZDim;
													WorkAreaState[j].Supporto.ZDim_Ext1        		:= WorkAreaState[j].Supporto.ZDim + 20;
													//Lo que HABIA	
													//WorkAreaOffset[j].Y 							:= HMI_OffsetDepositoLastra.Y180 ;
													//Mod 25/&/2025	  
													WorkAreaOffset[NumPostazioneDeposito].Y 		:= ActualPickingListFromHMI[IdxLista].SupportVertBundle.YDim-ActualPickingListFromHMI[IdxLista].SupportVertBundle.DimBaseUtile -40 ;			
												(* Se ho un A_Frame *)	  
												A_FRAME_VERT:  						
													//WorkAreaState[j].P := ElementiDaDepositare;
													WorkAreaState[j].Supporto.Code 					:= ActualPickingListFromHMI[IdxLista].SupportVertCav.Code;
													WorkAreaState[j].Supporto.DimBaseUtile		 	:= ActualPickingListFromHMI[IdxLista].SupportVertCav.DimBaseUtile;
													WorkAreaState[j].Supporto.AltezzaDenteRitenuta 	:= ActualPickingListFromHMI[IdxLista].SupportVertCav.ZDim+20;
													WorkAreaState[j].Supporto.DimVertice 			:= ActualPickingListFromHMI[IdxLista].SupportVertCav.DimVertice;
													WorkAreaState[j].Supporto.HMAX 					:= ActualPickingListFromHMI[IdxLista].SupportVertCav.HMAX;
													WorkAreaState[j].Supporto.Tipologia 			:= CAVALLETTO;//ActualPickingListFromHMI.SupportVertCav.Tipologia;
													WorkAreaState[j].Supporto.XDim 					:= ActualPickingListFromHMI[IdxLista].SupportVertCav.XDim;
													WorkAreaState[j].Supporto.YDim 					:= ActualPickingListFromHMI[IdxLista].SupportVertCav.YDim;
													WorkAreaState[j].Supporto.ZDim 					:= ActualPickingListFromHMI[IdxLista].SupportVertCav.ZDim;
													WorkAreaState[j].Supporto.ZDim_Ext1        		:= WorkAreaState[j].Supporto.ZDim + 20;		
													WorkAreaOffset[j].Y 							:= OFFSET_POSTAZIONE_LEGNO + ActualPickingListFromHMI[IdxLista].SupportVertCav.YDim/2;//ATTENZIONE!!! per poter lavorare in centro con i supporti pari, questa misura è la distanza tra il riscontro bundle verticale e il centro postazione PARI
											   		CoordenadaPasillo0_Y := WorkArea[j].Y +  WorkAreaOffset[j].Y  - Dimensioni_Pinza.Spessore - INGOMBRO_RISCONTRO_BUNDLE - WorkAreaState[j].Supporto.YDim /2 ;
													CoordenadaPasillo180_Y := WorkArea[j].Y + WorkAreaState[j].Supporto.YDim /2 + WorkAreaOffset[j].Y  + Dimensioni_Pinza.Spessore + INGOMBRO_RISCONTRO_FRAME  ;	
											END_CASE	
											WorkAreaProductionList[j].Support := HMI_Formatura.HMI_Forming_Supporto; 
										END_IF
									END_IF     
									TFClearApprendimento(ADR(WorkAreaState[j].Apprendimento));//Azzeramento apprendimento 
								END_FOR
								EXIT; 
							(* Se ho un telaio in piano *)	 
							TELAIO_PIANO:	
								WorkAreaState[NumPostazioneDeposito].Supporto.Code 						:= ActualPickingListFromHMI[IdxLista].SupportPianoFerro.Code;
								WorkAreaState[NumPostazioneDeposito].Supporto.AltezzaDenteRitenuta 		:= ActualPickingListFromHMI[IdxLista].SupportPianoFerro.DimBaseUtile;
								WorkAreaState[NumPostazioneDeposito].Supporto.DimVertice 				:= ActualPickingListFromHMI[IdxLista].SupportPianoFerro.DimVertice;
								WorkAreaState[NumPostazioneDeposito].Supporto.HMAX 						:= ActualPickingListFromHMI[IdxLista].SupportPianoFerro.HMAX;
								WorkAreaState[NumPostazioneDeposito].Supporto.Tipologia 				:= CASSA_STANDARD;//ActualPickingListFromHMI.Support.Tipologia;
								WorkAreaState[NumPostazioneDeposito].Supporto.XDim 						:= ActualPickingListFromHMI[IdxLista].SupportPianoFerro.XDim;
								WorkAreaState[NumPostazioneDeposito].Supporto.YDim 						:= ActualPickingListFromHMI[IdxLista].SupportPianoFerro.YDim;
								WorkAreaState[NumPostazioneDeposito].Supporto.ZDim 						:= ActualPickingListFromHMI[IdxLista].SupportPianoFerro.ZDim;
								WorkAreaOffset[NumPostazioneDeposito].Y 								:= OFFSET_POSTAZIONE_TELAIO - ActualPickingListFromHMI[IdxLista].SupportPianoFerro.YDim/2;//ATTENZIONE!!! per poter lavorare in centro con i supporti pari, questa misura è la distanza tra il riscontro bundle verticale e il centro postazione PARI
								CASE HMI_WorkAreaDataPicking[NumPostazioneDeposito].Typology OF
									LEGNO_PIANO:
										 		WorkAreaProductionList[NumPostazioneDeposito].Support := WorkAreaState[NumPostazioneDeposito].Supporto;
												WorkAreaProductionList[NumPostazioneDeposito].Support.Tipologia	:= e_Tipo_Pallet.CASSA_STANDARD; 
									TELAIO_PIANO:
										 		WorkAreaProductionList[NumPostazioneDeposito].Support := WorkAreaState[NumPostazioneDeposito].Supporto;
												WorkAreaProductionList[NumPostazioneDeposito].Support.Tipologia	:= e_Tipo_Pallet.CASSA_STANDARD; 
									BUNDLE_VERT:
										 		WorkAreaProductionList[NumPostazioneDeposito].Support := WorkAreaState[NumPostazioneDeposito].Supporto;
												WorkAreaProductionList[NumPostazioneDeposito].Support.Tipologia	:= e_Tipo_Pallet.BUNDLE; 
									A_FRAME_VERT:
										 		WorkAreaProductionList[NumPostazioneDeposito].Support := WorkAreaState[NumPostazioneDeposito].Supporto;
												WorkAreaProductionList[NumPostazioneDeposito].Support.Tipologia	:= e_Tipo_Pallet.CAVALLETTO; 
								END_CASE
								
